   instKP8BtnAct.old.kp8Config[29].activate[5] := TRUE;
   instKP8BtnAct.old.kp8Config[29].activate[6] := TRUE;
   instKP8BtnAct.old.kp8Config[29].activate[7] := TRUE;
   instKP8BtnAct.old.kp8Config[29].colorOn1[0] := 'off';
   instKP8BtnAct.old.kp8Config[29].colorOn1[1] := 'yellow';
   instKP8BtnAct.old.kp8Config[29].colorOn1[2] := 'yellow';
   instKP8BtnAct.old.kp8Config[29].colorOn1[3] := 'yellow';
   instKP8BtnAct.old.kp8Config[29].colorOn1[4] := 'off';
   instKP8BtnAct.old.kp8Config[29].colorOn1[5] := 'yellow';
   instKP8BtnAct.old.kp8Config[29].colorOn1[6] := 'yellow';
   instKP8BtnAct.old.kp8Config[29].colorOn1[7] := 'yellow';
   instKP8BtnAct.old.kp8Config[29].colorOn2[0] := 'off';
   instKP8BtnAct.old.kp8Config[29].colorOn2[4] := 'off';
   instKP8BtnAct.old.kp8Config[29].colorOff[0] := 'off';
   instKP8BtnAct.old.kp8Config[29].colorOff[1] := 'green';
   instKP8BtnAct.old.kp8Config[29].colorOff[2] := 'green';
   instKP8BtnAct.old.kp8Config[29].colorOff[3] := 'green';
   instKP8BtnAct.old.kp8Config[29].colorOff[4] := 'off';
   instKP8BtnAct.old.kp8Config[29].colorOff[5] := 'green';
   instKP8BtnAct.old.kp8Config[29].colorOff[6] := 'green';
   instKP8BtnAct.old.kp8Config[29].colorOff[7] := 'green';
   instKP8BtnAct.old.kp8Config[29].mode[1] := TRUE;
   instKP8BtnAct.old.kp8Config[29].mode[2] := TRUE;
   instKP8BtnAct.old.kp8Config[29].mode[3] := TRUE;
   instKP8BtnAct.old.kp8Config[29].mode[5] := TRUE;
   instKP8BtnAct.old.kp8Config[29].mode[6] := TRUE;
   instKP8BtnAct.old.kp8Config[29].mode[7] := TRUE;
   instKP8BtnAct.old.kp8Config[30].activate[7] := TRUE;
   instKP8BtnAct.old.kp8Config[30].colorOn1[0] := 'off';
   instKP8BtnAct.old.kp8Config[30].colorOn1[1] := 'off';
   instKP8BtnAct.old.kp8Config[30].colorOn1[2] := 'off';
   instKP8BtnAct.old.kp8Config[30].colorOn1[3] := 'off';
   instKP8BtnAct.old.kp8Config[30].colorOn1[4] := 'off';
   instKP8BtnAct.old.kp8Config[30].colorOn1[5] := 'off';
   instKP8BtnAct.old.kp8Config[30].colorOn1[6] := 'off';
   instKP8BtnAct.old.kp8Config[30].colorOn1[7] := 'yellow';
   instKP8BtnAct.old.kp8Config[30].colorOn2[0] := 'off';
   instKP8BtnAct.old.kp8Config[30].colorOn2[1] := 'off';
   instKP8BtnAct.old.kp8Config[30].colorOn2[2] := 'off';
   instKP8BtnAct.old.kp8Config[30].colorOn2[3] := 'off';
   instKP8BtnAct.old.kp8Config[30].colorOn2[4] := 'off';
   instKP8BtnAct.old.kp8Config[30].colorOn2[5] := 'off';
   instKP8BtnAct.old.kp8Config[30].colorOn2[6] := 'off';
   instKP8BtnAct.old.kp8Config[30].colorOff[0] := 'off';
   instKP8BtnAct.old.kp8Config[30].colorOff[1] := 'off';
   instKP8BtnAct.old.kp8Config[30].colorOff[2] := 'off';
   instKP8BtnAct.old.kp8Config[30].colorOff[3] := 'off';
   instKP8BtnAct.old.kp8Config[30].colorOff[4] := 'off';
   instKP8BtnAct.old.kp8Config[30].colorOff[5] := 'off';
   instKP8BtnAct.old.kp8Config[30].colorOff[6] := 'off';
   instKP8BtnAct.old.kp8Config[30].colorOff[7] := 'green';
   instKP8BtnAct.old.kp8Config[30].mode[7] := TRUE;
   instKP8BtnAct.old.kp8Config[31].activate[3] := TRUE;
   instKP8BtnAct.old.kp8Config[31].activate[7] := TRUE;
   instKP8BtnAct.old.kp8Config[31].colorOn1[0] := 'off';
   instKP8BtnAct.old.kp8Config[31].colorOn1[1] := 'off';
   instKP8BtnAct.old.kp8Config[31].colorOn1[2] := 'off';
   instKP8BtnAct.old.kp8Config[31].colorOn1[3] := 'yellow';
   instKP8BtnAct.old.kp8Config[31].colorOn1[4] := 'off';
   instKP8BtnAct.old.kp8Config[31].colorOn1[5] := 'off';
   instKP8BtnAct.old.kp8Config[31].colorOn1[6] := 'off';
   instKP8BtnAct.old.kp8Config[31].colorOn1[7] := 'yellow';
   instKP8BtnAct.old.kp8Config[31].colorOn2[0] := 'off';
   instKP8BtnAct.old.kp8Config[31].colorOn2[1] := 'off';
   instKP8BtnAct.old.kp8Config[31].colorOn2[2] := 'off';
   instKP8BtnAct.old.kp8Config[31].colorOn2[4] := 'off';
   instKP8BtnAct.old.kp8Config[31].colorOn2[5] := 'off';
   instKP8BtnAct.old.kp8Config[31].colorOn2[6] := 'off';
   instKP8BtnAct.old.kp8Config[31].colorOff[0] := 'off';
   instKP8BtnAct.old.kp8Config[31].colorOff[1] := 'off';
   instKP8BtnAct.old.kp8Config[31].colorOff[2] := 'off';
   instKP8BtnAct.old.kp8Config[31].colorOff[3] := 'green';
   instKP8BtnAct.old.kp8Config[31].colorOff[4] := 'off';
   instKP8BtnAct.old.kp8Config[31].colorOff[5] := 'off';
   instKP8BtnAct.old.kp8Config[31].colorOff[6] := 'off';
   instKP8BtnAct.old.kp8Config[31].colorOff[7] := 'green';
   instKP8BtnAct.old.kp8Config[31].mode[3] := TRUE;
   instKP8BtnAct.old.kp8Config[31].mode[7] := TRUE;
   instKP8BtnAct.old.kp8Config[32].activate[7] := TRUE;
   instKP8BtnAct.old.kp8Config[32].colorOn1[0] := 'off';
   instKP8BtnAct.old.kp8Config[32].colorOn1[1] := 'off';
   instKP8BtnAct.old.kp8Config[32].colorOn1[2] := 'off';
   instKP8BtnAct.old.kp8Config[32].colorOn1[3] := 'off';
   instKP8BtnAct.old.kp8Config[32].colorOn1[4] := 'off';
   instKP8BtnAct.old.kp8Config[32].colorOn1[5] := 'off';
   instKP8BtnAct.old.kp8Config[32].colorOn1[6] := 'off';
   instKP8BtnAct.old.kp8Config[32].colorOn1[7] := 'yellow';
   instKP8BtnAct.old.kp8Config[32].colorOn2[0] := 'off';
   instKP8BtnAct.old.kp8Config[32].colorOn2[1] := 'off';
   instKP8BtnAct.old.kp8Config[32].colorOn2[2] := 'off';
   instKP8BtnAct.old.kp8Config[32].colorOn2[3] := 'off';
   instKP8BtnAct.old.kp8Config[32].colorOn2[4] := 'off';
   instKP8BtnAct.old.kp8Config[32].colorOn2[5] := 'off';
   instKP8BtnAct.old.kp8Config[32].colorOn2[6] := 'off';
   instKP8BtnAct.old.kp8Config[32].colorOff[0] := 'off';
   instKP8BtnAct.old.kp8Config[32].colorOff[1] := 'off';
   instKP8BtnAct.old.kp8Config[32].colorOff[2] := 'off';
   instKP8BtnAct.old.kp8Config[32].colorOff[3] := 'off';
   instKP8BtnAct.old.kp8Config[32].colorOff[4] := 'off';
   instKP8BtnAct.old.kp8Config[32].colorOff[5] := 'off';
   instKP8BtnAct.old.kp8Config[32].colorOff[6] := 'off';
   instKP8BtnAct.old.kp8Config[32].colorOff[7] := 'green';
   instKP8BtnAct.old.kp8Config[32].mode[7] := TRUE;
   instKP8BtnAct.old.kp8Config[33].activate[7] := TRUE;
   instKP8BtnAct.old.kp8Config[33].colorOn1[0] := 'off';
   instKP8BtnAct.old.kp8Config[33].colorOn1[1] := 'off';
   instKP8BtnAct.old.kp8Config[33].colorOn1[2] := 'off';
   instKP8BtnAct.old.kp8Config[33].colorOn1[3] := 'off';
   instKP8BtnAct.old.kp8Config[33].colorOn1[4] := 'off';
   instKP8BtnAct.old.kp8Config[33].colorOn1[5] := 'off';
   instKP8BtnAct.old.kp8Config[33].colorOn1[6] := 'off';
   instKP8BtnAct.old.kp8Config[33].colorOn1[7] := 'yellow';
   instKP8BtnAct.old.kp8Config[33].colorOn2[0] := 'off';
   instKP8BtnAct.old.kp8Config[33].colorOn2[1] := 'off';
   instKP8BtnAct.old.kp8Config[33].colorOn2[2] := 'off';
   instKP8BtnAct.old.kp8Config[33].colorOn2[3] := 'off';
   instKP8BtnAct.old.kp8Config[33].colorOn2[4] := 'off';
   instKP8BtnAct.old.kp8Config[33].colorOn2[5] := 'off';
   instKP8BtnAct.old.kp8Config[33].colorOn2[6] := 'off';
   instKP8BtnAct.old.kp8Config[33].colorOff[0] := 'off';
   instKP8BtnAct.old.kp8Config[33].colorOff[1] := 'off';
   instKP8BtnAct.old.kp8Config[33].colorOff[2] := 'off';
   instKP8BtnAct.old.kp8Config[33].colorOff[3] := 'off';
   instKP8BtnAct.old.kp8Config[33].colorOff[4] := 'off';
   instKP8BtnAct.old.kp8Config[33].colorOff[5] := 'off';
   instKP8BtnAct.old.kp8Config[33].colorOff[6] := 'off';
   instKP8BtnAct.old.kp8Config[33].colorOff[7] := 'green';
   instKP8BtnAct.old.kp8Config[33].mode[7] := TRUE;
   instKP8BtnAct.old.kp8Config[34].activate[3] := TRUE;
   instKP8BtnAct.old.kp8Config[34].activate[7] := TRUE;
   instKP8BtnAct.old.kp8Config[34].colorOn1[0] := 'off';
   instKP8BtnAct.old.kp8Config[34].colorOn1[1] := 'off';
   instKP8BtnAct.old.kp8Config[34].colorOn1[2] := 'off';
   instKP8BtnAct.old.kp8Config[34].colorOn1[3] := 'yellow';
   instKP8BtnAct.old.kp8Config[34].colorOn1[4] := 'off';
   instKP8BtnAct.old.kp8Config[34].colorOn1[5] := 'off';
   instKP8BtnAct.old.kp8Config[34].colorOn1[6] := 'off';
   instKP8BtnAct.old.kp8Config[34].colorOn1[7] := 'yellow';
   instKP8BtnAct.old.kp8Config[34].colorOn2[0] := 'off';
   instKP8BtnAct.old.kp8Config[34].colorOn2[1] := 'off';
   instKP8BtnAct.old.kp8Config[34].colorOn2[2] := 'off';
   instKP8BtnAct.old.kp8Config[34].colorOn2[4] := 'off';
   instKP8BtnAct.old.kp8Config[34].colorOn2[5] := 'off';
   instKP8BtnAct.old.kp8Config[34].colorOn2[6] := 'off';
   instKP8BtnAct.old.kp8Config[34].colorOff[0] := 'off';
   instKP8BtnAct.old.kp8Config[34].colorOff[1] := 'off';
   instKP8BtnAct.old.kp8Config[34].colorOff[2] := 'off';
   instKP8BtnAct.old.kp8Config[34].colorOff[3] := 'green';
   instKP8BtnAct.old.kp8Config[34].colorOff[4] := 'off';
   instKP8BtnAct.old.kp8Config[34].colorOff[5] := 'off';
   instKP8BtnAct.old.kp8Config[34].colorOff[6] := 'off';
   instKP8BtnAct.old.kp8Config[34].colorOff[7] := 'green';
   instKP8BtnAct.old.kp8Config[34].mode[3] := TRUE;
   instKP8BtnAct.old.kp8Config[34].mode[7] := TRUE;
   instKP8BtnAct.old.kp8Config[35].activate[3] := TRUE;
   instKP8BtnAct.old.kp8Config[35].activate[7] := TRUE;
   instKP8BtnAct.old.kp8Config[35].colorOn1[0] := 'off';
   instKP8BtnAct.old.kp8Config[35].colorOn1[1] := 'off';
   instKP8BtnAct.old.kp8Config[35].colorOn1[2] := 'off';
   instKP8BtnAct.old.kp8Config[35].colorOn1[3] := 'yellow';
   instKP8BtnAct.old.kp8Config[35].colorOn1[4] := 'off';
   instKP8BtnAct.old.kp8Config[35].colorOn1[5] := 'off';
   instKP8BtnAct.old.kp8Config[35].colorOn1[6] := 'off';
   instKP8BtnAct.old.kp8Config[35].colorOn1[7] := 'yellow';
   instKP8BtnAct.old.kp8Config[35].colorOn2[0] := 'off';
   instKP8BtnAct.old.kp8Config[35].colorOn2[1] := 'off';
   instKP8BtnAct.old.kp8Config[35].colorOn2[2] := 'off';
   instKP8BtnAct.old.kp8Config[35].colorOn2[4] := 'off';
   instKP8BtnAct.old.kp8Config[35].colorOn2[5] := 'off';
   instKP8BtnAct.old.kp8Config[35].colorOn2[6] := 'off';
   instKP8BtnAct.old.kp8Config[35].colorOff[0] := 'off';
   instKP8BtnAct.old.kp8Config[35].colorOff[1] := 'off';
   instKP8BtnAct.old.kp8Config[35].colorOff[2] := 'off';
   instKP8BtnAct.old.kp8Config[35].colorOff[3] := 'green';
   instKP8BtnAct.old.kp8Config[35].colorOff[4] := 'off';
   instKP8BtnAct.old.kp8Config[35].colorOff[5] := 'off';
   instKP8BtnAct.old.kp8Config[35].colorOff[6] := 'off';
   instKP8BtnAct.old.kp8Config[35].colorOff[7] := 'green';
   instKP8BtnAct.old.kp8Config[35].mode[3] := TRUE;
   instKP8BtnAct.old.kp8Config[35].mode[7] := TRUE;
   instKP8BtnAct.old.kp8Config[36].activate[3] := TRUE;
   instKP8BtnAct.old.kp8Config[36].activate[7] := TRUE;
   instKP8BtnAct.old.kp8Config[36].colorOn1[0] := 'off';
   instKP8BtnAct.old.kp8Config[36].colorOn1[1] := 'off';
   instKP8BtnAct.old.kp8Config[36].colorOn1[2] := 'off';
   instKP8BtnAct.old.kp8Config[36].colorOn1[3] := 'yellow';
   instKP8BtnAct.old.kp8Config[36].colorOn1[4] := 'off';
   instKP8BtnAct.old.kp8Config[36].colorOn1[5] := 'off';
   instKP8BtnAct.old.kp8Config[36].colorOn1[6] := 'off';
   instKP8BtnAct.old.kp8Config[36].colorOn1[7] := 'yellow';
   instKP8BtnAct.old.kp8Config[36].colorOn2[0] := 'off';
   instKP8BtnAct.old.kp8Config[36].colorOn2[1] := 'off';
   instKP8BtnAct.old.kp8Config[36].colorOn2[2] := 'off';
   instKP8BtnAct.old.kp8Config[36].colorOn2[4] := 'off';
   instKP8BtnAct.old.kp8Config[36].colorOn2[5] := 'off';
   instKP8BtnAct.old.kp8Config[36].colorOn2[6] := 'off';
   instKP8BtnAct.old.kp8Config[36].colorOff[0] := 'off';
   instKP8BtnAct.old.kp8Config[36].colorOff[1] := 'off';
   instKP8BtnAct.old.kp8Config[36].colorOff[2] := 'off';
   instKP8BtnAct.old.kp8Config[36].colorOff[3] := 'green';
   instKP8BtnAct.old.kp8Config[36].colorOff[4] := 'off';
   instKP8BtnAct.old.kp8Config[36].colorOff[5] := 'off';
   instKP8BtnAct.old.kp8Config[36].colorOff[6] := 'off';
   instKP8BtnAct.old.kp8Config[36].colorOff[7] := 'green';
   instKP8BtnAct.old.kp8Config[36].mode[3] := TRUE;
   instKP8BtnAct.old.kp8Config[36].mode[7] := TRUE;
   instKP8BtnAct.old.kp8Config[37].activate[3] := TRUE;
   instKP8BtnAct.old.kp8Config[37].activate[7] := TRUE;
   instKP8BtnAct.old.kp8Config[37].colorOn1[0] := 'off';
   instKP8BtnAct.old.kp8Config[37].colorOn1[1] := 'off';
   instKP8BtnAct.old.kp8Config[37].colorOn1[2] := 'off';
   instKP8BtnAct.old.kp8Config[37].colorOn1[3] := 'yellow';
   instKP8BtnAct.old.kp8Config[37].colorOn1[4] := 'off';
   instKP8BtnAct.old.kp8Config[37].colorOn1[5] := 'off';
   instKP8BtnAct.old.kp8Config[37].colorOn1[6] := 'off';
   instKP8BtnAct.old.kp8Config[37].colorOn1[7] := 'yellow';
   instKP8BtnAct.old.kp8Config[37].colorOn2[0] := 'off';
   instKP8BtnAct.old.kp8Config[37].colorOn2[1] := 'off';
   instKP8BtnAct.old.kp8Config[37].colorOn2[2] := 'off';
   instKP8BtnAct.old.kp8Config[37].colorOn2[4] := 'off';
   instKP8BtnAct.old.kp8Config[37].colorOn2[5] := 'off';
   instKP8BtnAct.old.kp8Config[37].colorOn2[6] := 'off';
   instKP8BtnAct.old.kp8Config[37].colorOff[0] := 'off';
   instKP8BtnAct.old.kp8Config[37].colorOff[1] := 'off';
   instKP8BtnAct.old.kp8Config[37].colorOff[2] := 'off';
   instKP8BtnAct.old.kp8Config[37].colorOff[3] := 'green';
   instKP8BtnAct.old.kp8Config[37].colorOff[4] := 'off';
   instKP8BtnAct.old.kp8Config[37].colorOff[5] := 'off';
   instKP8BtnAct.old.kp8Config[37].colorOff[6] := 'off';
   instKP8BtnAct.old.kp8Config[37].colorOff[7] := 'green';
   instKP8BtnAct.old.kp8Config[37].mode[3] := TRUE;
   instKP8BtnAct.old.kp8Config[37].mode[7] := TRUE;
   instKP8BtnAct.old.kp8Config[38].activate[7] := TRUE;
   instKP8BtnAct.old.kp8Config[38].colorOn1[0] := 'off';
   instKP8BtnAct.old.kp8Config[38].colorOn1[1] := 'off';
   instKP8BtnAct.old.kp8Config[38].colorOn1[2] := 'off';
   instKP8BtnAct.old.kp8Config[38].colorOn1[3] := 'off';
   instKP8BtnAct.old.kp8Config[38].colorOn1[4] := 'off';
   instKP8BtnAct.old.kp8Config[38].colorOn1[5] := 'off';
   instKP8BtnAct.old.kp8Config[38].colorOn1[6] := 'off';
   instKP8BtnAct.old.kp8Config[38].colorOn1[7] := 'yellow';
   instKP8BtnAct.old.kp8Config[38].colorOn2[0] := 'off';
   instKP8BtnAct.old.kp8Config[38].colorOn2[1] := 'off';
   instKP8BtnAct.old.kp8Config[38].colorOn2[2] := 'off';
   instKP8BtnAct.old.kp8Config[38].colorOn2[3] := 'off';
   instKP8BtnAct.old.kp8Config[38].colorOn2[4] := 'off';
   instKP8BtnAct.old.kp8Config[38].colorOn2[5] := 'off';
   instKP8BtnAct.old.kp8Config[38].colorOn2[6] := 'off';
   instKP8BtnAct.old.kp8Config[38].colorOff[0] := 'off';
   instKP8BtnAct.old.kp8Config[38].colorOff[1] := 'off';
   instKP8BtnAct.old.kp8Config[38].colorOff[2] := 'off';
   instKP8BtnAct.old.kp8Config[38].colorOff[3] := 'off';
   instKP8BtnAct.old.kp8Config[38].colorOff[4] := 'off';
   instKP8BtnAct.old.kp8Config[38].colorOff[5] := 'off';
   instKP8BtnAct.old.kp8Config[38].colorOff[6] := 'off';
   instKP8BtnAct.old.kp8Config[38].colorOff[7] := 'green';
   instKP8BtnAct.old.kp8Config[38].mode[7] := TRUE;
   instKP8Drvs[0].btn0ColorOn1 := 'off';
   instKP8Drvs[0].btn0ColorOn2 := 'off';
   instKP8Drvs[0].btn0ColorOff := 'off';
   instKP8Drvs[0].btn1ColorOn1 := 'off';
   instKP8Drvs[0].btn1ColorOn2 := 'off';
   instKP8Drvs[0].btn1ColorOff := 'off';
   instKP8Drvs[0].btn2ColorOn1 := 'off';
   instKP8Drvs[0].btn2ColorOn2 := 'off';
   instKP8Drvs[0].btn2ColorOff := 'off';
   instKP8Drvs[0].btn3Activate := TRUE;
   instKP8Drvs[0].btn3Mode := TRUE;
   instKP8Drvs[0].btn3ColorOn1 := 'yellow';
   instKP8Drvs[0].btn3ColorOff := 'green';
   instKP8Drvs[0].btn4ColorOn1 := 'off';
   instKP8Drvs[0].btn4ColorOn2 := 'off';
   instKP8Drvs[0].btn4ColorOff := 'off';
   instKP8Drvs[0].btn5ColorOn1 := 'off';
   instKP8Drvs[0].btn5ColorOn2 := 'off';
   instKP8Drvs[0].btn5ColorOff := 'off';
   instKP8Drvs[0].btn6ColorOn1 := 'off';
   instKP8Drvs[0].btn6ColorOn2 := 'off';
   instKP8Drvs[0].btn6ColorOff := 'off';
   instKP8Drvs[0].btn7Activate := TRUE;
   instKP8Drvs[0].btn7Mode := TRUE;
   instKP8Drvs[0].btn7ColorOn1 := 'yellow';
   instKP8Drvs[0].btn7ColorOff := 'green';
   instKP8Drvs[0].btnColorsOut := 16#0088_0000;
   instKP8Drvs[0].i1 := 8;
   instKP8Drvs[0].i2 := 8;
   instKP8Drvs[0].btnActivateInt[3] := TRUE;
   instKP8Drvs[0].btnActivateInt[7] := TRUE;
   instKP8Drvs[0].btnClrMskOffInt[0] := 16#0000_0000;
   instKP8Drvs[0].btnClrMskOffInt[1] := 16#0000_0000;
   instKP8Drvs[0].btnClrMskOffInt[2] := 16#0000_0000;
   instKP8Drvs[0].btnClrMskOffInt[3] := 16#0008_0000;
   instKP8Drvs[0].btnClrMskOffInt[4] := 16#0000_0000;
   instKP8Drvs[0].btnClrMskOffInt[5] := 16#0000_0000;
   instKP8Drvs[0].btnClrMskOffInt[6] := 16#0000_0000;
   instKP8Drvs[0].btnClrMskOffInt[7] := 16#0080_0000;
   instKP8Drvs[0].btnClrMskOn1Int[0] := 16#0000_0000;
   instKP8Drvs[0].btnClrMskOn1Int[1] := 16#0000_0000;
   instKP8Drvs[0].btnClrMskOn1Int[2] := 16#0000_0000;
   instKP8Drvs[0].btnClrMskOn1Int[3] := 16#0808_0000;
   instKP8Drvs[0].btnClrMskOn1Int[4] := 16#0000_0000;
   instKP8Drvs[0].btnClrMskOn1Int[5] := 16#0000_0000;
   instKP8Drvs[0].btnClrMskOn1Int[6] := 16#0000_0000;
   instKP8Drvs[0].btnClrMskOn1Int[7] := 16#8080_0000;
   instKP8Drvs[0].btnClrMskOn2Int[0] := 16#0000_0000;
   instKP8Drvs[0].btnClrMskOn2Int[1] := 16#0000_0000;
   instKP8Drvs[0].btnClrMskOn2Int[2] := 16#0000_0000;
   instKP8Drvs[0].btnClrMskOn2Int[3] := 16#0000_0000;
   instKP8Drvs[0].btnClrMskOn2Int[4] := 16#0000_0000;
   instKP8Drvs[0].btnClrMskOn2Int[5] := 16#0000_0000;
   instKP8Drvs[0].btnClrMskOn2Int[6] := 16#0000_0000;
   instKP8Drvs[0].btnClrMskOn2Int[7] := 16#0000_0000;
   instKP8Drvs[0].btnClrOffInt[0] := 'off';
   instKP8Drvs[0].btnClrOffInt[1] := 'off';
   instKP8Drvs[0].btnClrOffInt[2] := 'off';
   instKP8Drvs[0].btnClrOffInt[3] := 'green';
   instKP8Drvs[0].btnClrOffInt[4] := 'off';
   instKP8Drvs[0].btnClrOffInt[5] := 'off';
   instKP8Drvs[0].btnClrOffInt[6] := 'off';
   instKP8Drvs[0].btnClrOffInt[7] := 'green';
   instKP8Drvs[0].btnClrOn1Int[0] := 'off';
   instKP8Drvs[0].btnClrOn1Int[1] := 'off';
   instKP8Drvs[0].btnClrOn1Int[2] := 'off';
   instKP8Drvs[0].btnClrOn1Int[3] := 'yellow';
   instKP8Drvs[0].btnClrOn1Int[4] := 'off';
   instKP8Drvs[0].btnClrOn1Int[5] := 'off';
   instKP8Drvs[0].btnClrOn1Int[6] := 'off';
   instKP8Drvs[0].btnClrOn1Int[7] := 'yellow';
   instKP8Drvs[0].btnClrOn2Int[0] := 'off';
   instKP8Drvs[0].btnClrOn2Int[1] := 'off';
   instKP8Drvs[0].btnClrOn2Int[2] := 'off';
   instKP8Drvs[0].btnClrOn2Int[4] := 'off';
   instKP8Drvs[0].btnClrOn2Int[5] := 'off';
   instKP8Drvs[0].btnClrOn2Int[6] := 'off';
   instKP8Drvs[0].btnColors := 16#0088_0000;
   instKP8Drvs[0].btnModeInt[3] := TRUE;
   instKP8Drvs[0].btnModeInt[7] := TRUE;
   instKP8Drvs[1].btn0ColorOn1 := 'off';
   instKP8Drvs[1].btn0ColorOn2 := 'off';
   instKP8Drvs[1].btn0ColorOff := 'off';
   instKP8Drvs[1].btn1ColorOn1 := 'off';
   instKP8Drvs[1].btn1ColorOn2 := 'off';
   instKP8Drvs[1].btn1ColorOff := 'off';
   instKP8Drvs[1].btn2Activate := TRUE;
   instKP8Drvs[1].btn2Mode := TRUE;
   instKP8Drvs[1].btn2ColorOn1 := 'yellow';
   instKP8Drvs[1].btn2ColorOff := 'green';
   instKP8Drvs[1].btn3Activate := TRUE;
   instKP8Drvs[1].btn3Mode := TRUE;
   instKP8Drvs[1].btn3ColorOn1 := 'yellow';
   instKP8Drvs[1].btn3ColorOff := 'green';
   instKP8Drvs[1].btn4ColorOn1 := 'off';
   instKP8Drvs[1].btn4ColorOn2 := 'off';
   instKP8Drvs[1].btn4ColorOff := 'off';
   instKP8Drvs[1].btn5ColorOn1 := 'off';
   instKP8Drvs[1].btn5ColorOn2 := 'off';
   instKP8Drvs[1].btn5ColorOff := 'off';
   instKP8Drvs[1].btn6Activate := TRUE;
   instKP8Drvs[1].btn6Mode := TRUE;
   instKP8Drvs[1].btn6ColorOn1 := 'yellow';
   instKP8Drvs[1].btn6ColorOff := 'green';
   instKP8Drvs[1].btn7Activate := TRUE;
   instKP8Drvs[1].btn7Mode := TRUE;
   instKP8Drvs[1].btn7ColorOn1 := 'yellow';
   instKP8Drvs[1].btn7ColorOff := 'green';
   instKP8Drvs[1].btnColorsOut := 16#00CC_0000;
   instKP8Drvs[1].i1 := 8;
   instKP8Drvs[1].i2 := 8;
   instKP8Drvs[1].btnActivateInt[2] := TRUE;
   instKP8Drvs[1].btnActivateInt[3] := TRUE;
   instKP8Drvs[1].btnActivateInt[6] := TRUE;
   instKP8Drvs[1].btnActivateInt[7] := TRUE;
   instKP8Drvs[1].btnClrMskOffInt[0] := 16#0000_0000;
   instKP8Drvs[1].btnClrMskOffInt[1] := 16#0000_0000;
   instKP8Drvs[1].btnClrMskOffInt[2] := 16#0004_0000;
   instKP8Drvs[1].btnClrMskOffInt[3] := 16#0008_0000;
   instKP8Drvs[1].btnClrMskOffInt[4] := 16#0000_0000;
   instKP8Drvs[1].btnClrMskOffInt[5] := 16#0000_0000;
   instKP8Drvs[1].btnClrMskOffInt[6] := 16#0040_0000;
   instKP8Drvs[1].btnClrMskOffInt[7] := 16#0080_0000;
   instKP8Drvs[1].btnClrMskOn1Int[0] := 16#0000_0000;
   instKP8Drvs[1].btnClrMskOn1Int[1] := 16#0000_0000;
   instKP8Drvs[1].btnClrMskOn1Int[2] := 16#0404_0000;
   instKP8Drvs[1].btnClrMskOn1Int[3] := 16#0808_0000;
   instKP8Drvs[1].btnClrMskOn1Int[4] := 16#0000_0000;
   instKP8Drvs[1].btnClrMskOn1Int[5] := 16#0000_0000;
   instKP8Drvs[1].btnClrMskOn1Int[6] := 16#4040_0000;
   instKP8Drvs[1].btnClrMskOn1Int[7] := 16#8080_0000;
   instKP8Drvs[1].btnClrMskOn2Int[0] := 16#0000_0000;
   instKP8Drvs[1].btnClrMskOn2Int[1] := 16#0000_0000;
   instKP8Drvs[1].btnClrMskOn2Int[2] := 16#0000_0000;
   instKP8Drvs[1].btnClrMskOn2Int[3] := 16#0000_0000;
   instKP8Drvs[1].btnClrMskOn2Int[4] := 16#0000_0000;
   instKP8Drvs[1].btnClrMskOn2Int[5] := 16#0000_0000;
   instKP8Drvs[1].btnClrMskOn2Int[6] := 16#0000_0000;
   instKP8Drvs[1].btnClrMskOn2Int[7] := 16#0000_0000;
   instKP8Drvs[1].btnClrOffInt[0] := 'off';
   instKP8Drvs[1].btnClrOffInt[1] := 'off';
   instKP8Drvs[1].btnClrOffInt[2] := 'green';
   instKP8Drvs[1].btnClrOffInt[3] := 'green';
   instKP8Drvs[1].btnClrOffInt[4] := 'off';
   instKP8Drvs[1].btnClrOffInt[5] := 'off';
   instKP8Drvs[1].btnClrOffInt[6] := 'green';
   instKP8Drvs[1].btnClrOffInt[7] := 'green';
   instKP8Drvs[1].btnClrOn1Int[0] := 'off';
   instKP8Drvs[1].btnClrOn1Int[1] := 'off';
   instKP8Drvs[1].btnClrOn1Int[2] := 'yellow';
   instKP8Drvs[1].btnClrOn1Int[3] := 'yellow';
   instKP8Drvs[1].btnClrOn1Int[4] := 'off';
   instKP8Drvs[1].btnClrOn1Int[5] := 'off';
   instKP8Drvs[1].btnClrOn1Int[6] := 'yellow';
   instKP8Drvs[1].btnClrOn1Int[7] := 'yellow';
   instKP8Drvs[1].btnClrOn2Int[0] := 'off';
   instKP8Drvs[1].btnClrOn2Int[1] := 'off';
   instKP8Drvs[1].btnClrOn2Int[4] := 'off';
   instKP8Drvs[1].btnClrOn2Int[5] := 'off';
   instKP8Drvs[1].btnColors := 16#00CC_0000;
   instKP8Drvs[1].btnModeInt[2] := TRUE;
   instKP8Drvs[1].btnModeInt[3] := TRUE;
   instKP8Drvs[1].btnModeInt[6] := TRUE;
   instKP8Drvs[1].btnModeInt[7] := TRUE;
   instKP8Drvs[2].btn0ColorOn1 := 'off';
   instKP8Drvs[2].btn0ColorOn2 := 'off';
   instKP8Drvs[2].btn0ColorOff := 'off';
   instKP8Drvs[2].btn1Activate := TRUE;
   instKP8Drvs[2].btn1Mode := TRUE;
   instKP8Drvs[2].btn1ColorOn1 := 'yellow';
   instKP8Drvs[2].btn1ColorOff := 'green';
   instKP8Drvs[2].btn2Activate := TRUE;
   instKP8Drvs[2].btn2Mode := TRUE;
   instKP8Drvs[2].btn2ColorOn1 := 'yellow';
   instKP8Drvs[2].btn2ColorOff := 'green';
   instKP8Drvs[2].btn3Activate := TRUE;
   instKP8Drvs[2].btn3Mode := TRUE;
   instKP8Drvs[2].btn3ColorOn1 := 'yellow';
   instKP8Drvs[2].btn3ColorOff := 'green';
   instKP8Drvs[2].btn4ColorOn1 := 'off';
   instKP8Drvs[2].btn4ColorOn2 := 'off';
   instKP8Drvs[2].btn4ColorOff := 'off';
   instKP8Drvs[2].btn5Activate := TRUE;
   instKP8Drvs[2].btn5Mode := TRUE;
   instKP8Drvs[2].btn5ColorOn1 := 'yellow';
   instKP8Drvs[2].btn5ColorOff := 'green';
   instKP8Drvs[2].btn6Activate := TRUE;
   instKP8Drvs[2].btn6Mode := TRUE;
   instKP8Drvs[2].btn6ColorOn1 := 'yellow';
   instKP8Drvs[2].btn6ColorOff := 'green';
   instKP8Drvs[2].btn7Activate := TRUE;
   instKP8Drvs[2].btn7Mode := TRUE;
   instKP8Drvs[2].btn7ColorOn1 := 'yellow';
   instKP8Drvs[2].btn7ColorOff := 'green';
   instKP8Drvs[2].btnColorsOut := 16#00EE_0000;
   instKP8Drvs[2].i1 := 8;
   instKP8Drvs[2].i2 := 8;
   instKP8Drvs[2].btnActivateInt[1] := TRUE;
   instKP8Drvs[2].btnActivateInt[2] := TRUE;
   instKP8Drvs[2].btnActivateInt[3] := TRUE;
   instKP8Drvs[2].btnActivateInt[5] := TRUE;
   instKP8Drvs[2].btnActivateInt[6] := TRUE;
   instKP8Drvs[2].btnActivateInt[7] := TRUE;
   instKP8Drvs[2].btnClrMskOffInt[0] := 16#0000_0000;
   instKP8Drvs[2].btnClrMskOffInt[1] := 16#0002_0000;
   instKP8Drvs[2].btnClrMskOffInt[2] := 16#0004_0000;
   instKP8Drvs[2].btnClrMskOffInt[3] := 16#0008_0000;
   instKP8Drvs[2].btnClrMskOffInt[4] := 16#0000_0000;
   instKP8Drvs[2].btnClrMskOffInt[5] := 16#0020_0000;
   instKP8Drvs[2].btnClrMskOffInt[6] := 16#0040_0000;
   instKP8Drvs[2].btnClrMskOffInt[7] := 16#0080_0000;
   instKP8Drvs[2].btnClrMskOn1Int[0] := 16#0000_0000;
   instKP8Drvs[2].btnClrMskOn1Int[1] := 16#0202_0000;
   instKP8Drvs[2].btnClrMskOn1Int[2] := 16#0404_0000;
   instKP8Drvs[2].btnClrMskOn1Int[3] := 16#0808_0000;
   instKP8Drvs[2].btnClrMskOn1Int[4] := 16#0000_0000;
   instKP8Drvs[2].btnClrMskOn1Int[5] := 16#2020_0000;
   instKP8Drvs[2].btnClrMskOn1Int[6] := 16#4040_0000;
   instKP8Drvs[2].btnClrMskOn1Int[7] := 16#8080_0000;
   instKP8Drvs[2].btnClrMskOn2Int[0] := 16#0000_0000;
   instKP8Drvs[2].btnClrMskOn2Int[1] := 16#0000_0000;
   instKP8Drvs[2].btnClrMskOn2Int[2] := 16#0000_0000;
   instKP8Drvs[2].btnClrMskOn2Int[3] := 16#0000_0000;
   instKP8Drvs[2].btnClrMskOn2Int[4] := 16#0000_0000;
   instKP8Drvs[2].btnClrMskOn2Int[5] := 16#0000_0000;
   instKP8Drvs[2].btnClrMskOn2Int[6] := 16#0000_0000;
   instKP8Drvs[2].btnClrMskOn2Int[7] := 16#0000_0000;
   instKP8Drvs[2].btnClrOffInt[0] := 'off';
   instKP8Drvs[2].btnClrOffInt[1] := 'green';
   instKP8Drvs[2].btnClrOffInt[2] := 'green';
   instKP8Drvs[2].btnClrOffInt[3] := 'green';
   instKP8Drvs[2].btnClrOffInt[4] := 'off';
   instKP8Drvs[2].btnClrOffInt[5] := 'green';
   instKP8Drvs[2].btnClrOffInt[6] := 'green';
   instKP8Drvs[2].btnClrOffInt[7] := 'green';
   instKP8Drvs[2].btnClrOn1Int[0] := 'off';
   instKP8Drvs[2].btnClrOn1Int[1] := 'yellow';
   instKP8Drvs[2].btnClrOn1Int[2] := 'yellow';
   instKP8Drvs[2].btnClrOn1Int[3] := 'yellow';
   instKP8Drvs[2].btnClrOn1Int[4] := 'off';
   instKP8Drvs[2].btnClrOn1Int[5] := 'yellow';
   instKP8Drvs[2].btnClrOn1Int[6] := 'yellow';
   instKP8Drvs[2].btnClrOn1Int[7] := 'yellow';
   instKP8Drvs[2].btnClrOn2Int[0] := 'off';
   instKP8Drvs[2].btnClrOn2Int[4] := 'off';
   instKP8Drvs[2].btnColors := 16#00EE_0000;
   instKP8Drvs[2].btnModeInt[1] := TRUE;
   instKP8Drvs[2].btnModeInt[2] := TRUE;
   instKP8Drvs[2].btnModeInt[3] := TRUE;
   instKP8Drvs[2].btnModeInt[5] := TRUE;
   instKP8Drvs[2].btnModeInt[6] := TRUE;
   instKP8Drvs[2].btnModeInt[7] := TRUE;
   instKP8Drvs[3].btn0ColorOn1 := 'off';
   instKP8Drvs[3].btn0ColorOn2 := 'off';
   instKP8Drvs[3].btn0ColorOff := 'off';
   instKP8Drvs[3].btn1Activate := TRUE;
   instKP8Drvs[3].btn1Mode := TRUE;
   instKP8Drvs[3].btn1ColorOn1 := 'yellow';
   instKP8Drvs[3].btn1ColorOff := 'green';
   instKP8Drvs[3].btn2Activate := TRUE;
   instKP8Drvs[3].btn2Mode := TRUE;
   instKP8Drvs[3].btn2ColorOn1 := 'yellow';
   instKP8Drvs[3].btn2ColorOff := 'green';
   instKP8Drvs[3].btn3Activate := TRUE;
   instKP8Drvs[3].btn3Mode := TRUE;
   instKP8Drvs[3].btn3ColorOn1 := 'yellow';
   instKP8Drvs[3].btn3ColorOff := 'green';
   instKP8Drvs[3].btn4ColorOn1 := 'off';
   instKP8Drvs[3].btn4ColorOn2 := 'off';
   instKP8Drvs[3].btn4ColorOff := 'off';
   instKP8Drvs[3].btn5Activate := TRUE;
   instKP8Drvs[3].btn5Mode := TRUE;
   instKP8Drvs[3].btn5ColorOn1 := 'yellow';
   instKP8Drvs[3].btn5ColorOff := 'green';
   instKP8Drvs[3].btn6Activate := TRUE;
   instKP8Drvs[3].btn6Mode := TRUE;
   instKP8Drvs[3].btn6ColorOn1 := 'yellow';
   instKP8Drvs[3].btn6ColorOff := 'green';
   instKP8Drvs[3].btn7Activate := TRUE;
   instKP8Drvs[3].btn7Mode := TRUE;
   instKP8Drvs[3].btn7ColorOn1 := 'yellow';
   instKP8Drvs[3].btn7ColorOff := 'green';
   instKP8Drvs[3].btnColorsOut := 16#00EE_0000;
   instKP8Drvs[3].i1 := 8;
   instKP8Drvs[3].i2 := 8;
   instKP8Drvs[3].btnActivateInt[1] := TRUE;
   instKP8Drvs[3].btnActivateInt[2] := TRUE;
   instKP8Drvs[3].btnActivateInt[3] := TRUE;
   instKP8Drvs[3].btnActivateInt[5] := TRUE;
   instKP8Drvs[3].btnActivateInt[6] := TRUE;
   instKP8Drvs[3].btnActivateInt[7] := TRUE;
   instKP8Drvs[3].btnClrMskOffInt[0] := 16#0000_0000;
   instKP8Drvs[3].btnClrMskOffInt[1] := 16#0002_0000;
   instKP8Drvs[3].btnClrMskOffInt[2] := 16#0004_0000;
   instKP8Drvs[3].btnClrMskOffInt[3] := 16#0008_0000;
   instKP8Drvs[3].btnClrMskOffInt[4] := 16#0000_0000;
   instKP8Drvs[3].btnClrMskOffInt[5] := 16#0020_0000;
   instKP8Drvs[3].btnClrMskOffInt[6] := 16#0040_0000;
   instKP8Drvs[3].btnClrMskOffInt[7] := 16#0080_0000;
   instKP8Drvs[3].btnClrMskOn1Int[0] := 16#0000_0000;
   instKP8Drvs[3].btnClrMskOn1Int[1] := 16#0202_0000;
   instKP8Drvs[3].btnClrMskOn1Int[2] := 16#0404_0000;
   instKP8Drvs[3].btnClrMskOn1Int[3] := 16#0808_0000;
   instKP8Drvs[3].btnClrMskOn1Int[4] := 16#0000_0000;
   instKP8Drvs[3].btnClrMskOn1Int[5] := 16#2020_0000;
   instKP8Drvs[3].btnClrMskOn1Int[6] := 16#4040_0000;
   instKP8Drvs[3].btnClrMskOn1Int[7] := 16#8080_0000;
   instKP8Drvs[3].btnClrMskOn2Int[0] := 16#0000_0000;
   instKP8Drvs[3].btnClrMskOn2Int[1] := 16#0000_0000;
   instKP8Drvs[3].btnClrMskOn2Int[2] := 16#0000_0000;
   instKP8Drvs[3].btnClrMskOn2Int[3] := 16#0000_0000;
   instKP8Drvs[3].btnClrMskOn2Int[4] := 16#0000_0000;
   instKP8Drvs[3].btnClrMskOn2Int[5] := 16#0000_0000;
   instKP8Drvs[3].btnClrMskOn2Int[6] := 16#0000_0000;
   instKP8Drvs[3].btnClrMskOn2Int[7] := 16#0000_0000;
   instKP8Drvs[3].btnClrOffInt[0] := 'off';
   instKP8Drvs[3].btnClrOffInt[1] := 'green';
   instKP8Drvs[3].btnClrOffInt[2] := 'green';
   instKP8Drvs[3].btnClrOffInt[3] := 'green';
   instKP8Drvs[3].btnClrOffInt[4] := 'off';
   instKP8Drvs[3].btnClrOffInt[5] := 'green';
   instKP8Drvs[3].btnClrOffInt[6] := 'green';
   instKP8Drvs[3].btnClrOffInt[7] := 'green';
   instKP8Drvs[3].btnClrOn1Int[0] := 'off';
   instKP8Drvs[3].btnClrOn1Int[1] := 'yellow';
   instKP8Drvs[3].btnClrOn1Int[2] := 'yellow';
   instKP8Drvs[3].btnClrOn1Int[3] := 'yellow';
   instKP8Drvs[3].btnClrOn1Int[4] := 'off';
   instKP8Drvs[3].btnClrOn1Int[5] := 'yellow';
   instKP8Drvs[3].btnClrOn1Int[6] := 'yellow';
   instKP8Drvs[3].btnClrOn1Int[7] := 'yellow';
   instKP8Drvs[3].btnClrOn2Int[0] := 'off';
   instKP8Drvs[3].btnClrOn2Int[4] := 'off';
   instKP8Drvs[3].btnColors := 16#00EE_0000;
   instKP8Drvs[3].btnModeInt[1] := TRUE;
   instKP8Drvs[3].btnModeInt[2] := TRUE;
   instKP8Drvs[3].btnModeInt[3] := TRUE;
   instKP8Drvs[3].btnModeInt[5] := TRUE;
   instKP8Drvs[3].btnModeInt[6] := TRUE;
   instKP8Drvs[3].btnModeInt[7] := TRUE;
   instKP8Drvs[4].btn0ColorOn1 := 'off';
   instKP8Drvs[4].btn0ColorOn2 := 'off';
   instKP8Drvs[4].btn0ColorOff := 'off';
   instKP8Drvs[4].btn1ColorOn1 := 'off';
   instKP8Drvs[4].btn1ColorOn2 := 'off';
   instKP8Drvs[4].btn1ColorOff := 'off';
   instKP8Drvs[4].btn2ColorOn1 := 'off';
   instKP8Drvs[4].btn2ColorOn2 := 'off';
   instKP8Drvs[4].btn2ColorOff := 'off';
   instKP8Drvs[4].btn3ColorOn1 := 'off';
   instKP8Drvs[4].btn3ColorOn2 := 'off';
   instKP8Drvs[4].btn3ColorOff := 'off';
   instKP8Drvs[4].btn4ColorOn1 := 'off';
   instKP8Drvs[4].btn4ColorOn2 := 'off';
   instKP8Drvs[4].btn4ColorOff := 'off';
   instKP8Drvs[4].btn5ColorOn1 := 'off';
   instKP8Drvs[4].btn5ColorOn2 := 'off';
   instKP8Drvs[4].btn5ColorOff := 'off';
   instKP8Drvs[4].btn6ColorOn1 := 'off';
   instKP8Drvs[4].btn6ColorOn2 := 'off';
   instKP8Drvs[4].btn6ColorOff := 'off';
   instKP8Drvs[4].btn7Activate := TRUE;
   instKP8Drvs[4].btn7Mode := TRUE;
   instKP8Drvs[4].btn7ColorOn1 := 'yellow';
   instKP8Drvs[4].btn7ColorOff := 'green';
   instKP8Drvs[4].btnColorsOut := 16#0080_0000;
   instKP8Drvs[4].i1 := 8;
   instKP8Drvs[4].i2 := 8;
   instKP8Drvs[4].btnActivateInt[7] := TRUE;
   instKP8Drvs[4].btnClrMskOffInt[0] := 16#0000_0000;
   instKP8Drvs[4].btnClrMskOffInt[1] := 16#0000_0000;
   instKP8Drvs[4].btnClrMskOffInt[2] := 16#0000_0000;
   instKP8Drvs[4].btnClrMskOffInt[3] := 16#0000_0000;
   instKP8Drvs[4].btnClrMskOffInt[4] := 16#0000_0000;
   instKP8Drvs[4].btnClrMskOffInt[5] := 16#0000_0000;
   instKP8Drvs[4].btnClrMskOffInt[6] := 16#0000_0000;
   instKP8Drvs[4].btnClrMskOffInt[7] := 16#0080_0000;
   instKP8Drvs[4].btnClrMskOn1Int[0] := 16#0000_0000;
   instKP8Drvs[4].btnClrMskOn1Int[1] := 16#0000_0000;
   instKP8Drvs[4].btnClrMskOn1Int[2] := 16#0000_0000;
   instKP8Drvs[4].btnClrMskOn1Int[3] := 16#0000_0000;
   instKP8Drvs[4].btnClrMskOn1Int[4] := 16#0000_0000;
   instKP8Drvs[4].btnClrMskOn1Int[5] := 16#0000_0000;
   instKP8Drvs[4].btnClrMskOn1Int[6] := 16#0000_0000;
   instKP8Drvs[4].btnClrMskOn1Int[7] := 16#8080_0000;
   instKP8Drvs[4].btnClrMskOn2Int[0] := 16#0000_0000;
   instKP8Drvs[4].btnClrMskOn2Int[1] := 16#0000_0000;
   instKP8Drvs[4].btnClrMskOn2Int[2] := 16#0000_0000;
   instKP8Drvs[4].btnClrMskOn2Int[3] := 16#0000_0000;
   instKP8Drvs[4].btnClrMskOn2Int[4] := 16#0000_0000;
   instKP8Drvs[4].btnClrMskOn2Int[5] := 16#0000_0000;
   instKP8Drvs[4].btnClrMskOn2Int[6] := 16#0000_0000;
   instKP8Drvs[4].btnClrMskOn2Int[7] := 16#0000_0000;
   instKP8Drvs[4].btnClrOffInt[0] := 'off';
   instKP8Drvs[4].btnClrOffInt[1] := 'off';
   instKP8Drvs[4].btnClrOffInt[2] := 'off';
   instKP8Drvs[4].btnClrOffInt[3] := 'off';
   instKP8Drvs[4].btnClrOffInt[4] := 'off';
   instKP8Drvs[4].btnClrOffInt[5] := 'off';
   instKP8Drvs[4].btnClrOffInt[6] := 'off';
   instKP8Drvs[4].btnClrOffInt[7] := 'green';
   instKP8Drvs[4].btnClrOn1Int[0] := 'off';
   instKP8Drvs[4].btnClrOn1Int[1] := 'off';
   instKP8Drvs[4].btnClrOn1Int[2] := 'off';
   instKP8Drvs[4].btnClrOn1Int[3] := 'off';
   instKP8Drvs[4].btnClrOn1Int[4] := 'off';
   instKP8Drvs[4].btnClrOn1Int[5] := 'off';
   instKP8Drvs[4].btnClrOn1Int[6] := 'off';
   instKP8Drvs[4].btnClrOn1Int[7] := 'yellow';
   instKP8Drvs[4].btnClrOn2Int[0] := 'off';
   instKP8Drvs[4].btnClrOn2Int[1] := 'off';
   instKP8Drvs[4].btnClrOn2Int[2] := 'off';
   instKP8Drvs[4].btnClrOn2Int[3] := 'off';
   instKP8Drvs[4].btnClrOn2Int[4] := 'off';
   instKP8Drvs[4].btnClrOn2Int[5] := 'off';
   instKP8Drvs[4].btnClrOn2Int[6] := 'off';
   instKP8Drvs[4].btnColors := 16#0080_0000;
   instKP8Drvs[4].btnModeInt[7] := TRUE;
   instKP8Drvs[5].btn0ColorOn1 := 'off';
   instKP8Drvs[5].btn0ColorOn2 := 'off';
   instKP8Drvs[5].btn0ColorOff := 'off';
   instKP8Drvs[5].btn1Activate := TRUE;
   instKP8Drvs[5].btn1Mode := TRUE;
   instKP8Drvs[5].btn1ColorOn1 := 'yellow';
   instKP8Drvs[5].btn1ColorOff := 'green';
   instKP8Drvs[5].btn2Activate := TRUE;
   instKP8Drvs[5].btn2Mode := TRUE;
   instKP8Drvs[5].btn2ColorOn1 := 'yellow';
   instKP8Drvs[5].btn2ColorOff := 'green';
   instKP8Drvs[5].btn3Activate := TRUE;
   instKP8Drvs[5].btn3Mode := TRUE;
   instKP8Drvs[5].btn3ColorOn1 := 'yellow';
   instKP8Drvs[5].btn3ColorOff := 'green';
   instKP8Drvs[5].btn4ColorOn1 := 'off';
   instKP8Drvs[5].btn4ColorOn2 := 'off';
   instKP8Drvs[5].btn4ColorOff := 'off';
   instKP8Drvs[5].btn5Activate := TRUE;
   instKP8Drvs[5].btn5Mode := TRUE;
   instKP8Drvs[5].btn5ColorOn1 := 'yellow';
   instKP8Drvs[5].btn5ColorOff := 'green';
   instKP8Drvs[5].btn6Activate := TRUE;
   instKP8Drvs[5].btn6Mode := TRUE;
   instKP8Drvs[5].btn6ColorOn1 := 'yellow';
   instKP8Drvs[5].btn6ColorOff := 'green';
   instKP8Drvs[5].btn7Activate := TRUE;
   instKP8Drvs[5].btn7Mode := TRUE;
   instKP8Drvs[5].btn7ColorOn1 := 'yellow';
   instKP8Drvs[5].btn7ColorOff := 'green';
   instKP8Drvs[5].btnColorsOut := 16#00EE_0000;
   instKP8Drvs[5].i1 := 8;
   instKP8Drvs[5].i2 := 8;
   instKP8Drvs[5].btnActivateInt[1] := TRUE;
   instKP8Drvs[5].btnActivateInt[2] := TRUE;
   instKP8Drvs[5].btnActivateInt[3] := TRUE;
   instKP8Drvs[5].btnActivateInt[5] := TRUE;
   instKP8Drvs[5].btnActivateInt[6] := TRUE;
   instKP8Drvs[5].btnActivateInt[7] := TRUE;
   instKP8Drvs[5].btnClrMskOffInt[0] := 16#0000_0000;
   instKP8Drvs[5].btnClrMskOffInt[1] := 16#0002_0000;
   instKP8Drvs[5].btnClrMskOffInt[2] := 16#0004_0000;
   instKP8Drvs[5].btnClrMskOffInt[3] := 16#0008_0000;
   instKP8Drvs[5].btnClrMskOffInt[4] := 16#0000_0000;
   instKP8Drvs[5].btnClrMskOffInt[5] := 16#0020_0000;
   instKP8Drvs[5].btnClrMskOffInt[6] := 16#0040_0000;
   instKP8Drvs[5].btnClrMskOffInt[7] := 16#0080_0000;
   instKP8Drvs[5].btnClrMskOn1Int[0] := 16#0000_0000;
   instKP8Drvs[5].btnClrMskOn1Int[1] := 16#0202_0000;
   instKP8Drvs[5].btnClrMskOn1Int[2] := 16#0404_0000;
   instKP8Drvs[5].btnClrMskOn1Int[3] := 16#0808_0000;
   instKP8Drvs[5].btnClrMskOn1Int[4] := 16#0000_0000;
   instKP8Drvs[5].btnClrMskOn1Int[5] := 16#2020_0000;
   instKP8Drvs[5].btnClrMskOn1Int[6] := 16#4040_0000;
   instKP8Drvs[5].btnClrMskOn1Int[7] := 16#8080_0000;
   instKP8Drvs[5].btnClrMskOn2Int[0] := 16#0000_0000;
   instKP8Drvs[5].btnClrMskOn2Int[1] := 16#0000_0000;
   instKP8Drvs[5].btnClrMskOn2Int[2] := 16#0000_0000;
   instKP8Drvs[5].btnClrMskOn2Int[3] := 16#0000_0000;
   instKP8Drvs[5].btnClrMskOn2Int[4] := 16#0000_0000;
   instKP8Drvs[5].btnClrMskOn2Int[5] := 16#0000_0000;
   instKP8Drvs[5].btnClrMskOn2Int[6] := 16#0000_0000;
   instKP8Drvs[5].btnClrMskOn2Int[7] := 16#0000_0000;
   instKP8Drvs[5].btnClrOffInt[0] := 'off';
   instKP8Drvs[5].btnClrOffInt[1] := 'green';
   instKP8Drvs[5].btnClrOffInt[2] := 'green';
   instKP8Drvs[5].btnClrOffInt[3] := 'green';
   instKP8Drvs[5].btnClrOffInt[4] := 'off';
   instKP8Drvs[5].btnClrOffInt[5] := 'green';
   instKP8Drvs[5].btnClrOffInt[6] := 'green';
   instKP8Drvs[5].btnClrOffInt[7] := 'green';
   instKP8Drvs[5].btnClrOn1Int[0] := 'off';
   instKP8Drvs[5].btnClrOn1Int[1] := 'yellow';
   instKP8Drvs[5].btnClrOn1Int[2] := 'yellow';
   instKP8Drvs[5].btnClrOn1Int[3] := 'yellow';
   instKP8Drvs[5].btnClrOn1Int[4] := 'off';
   instKP8Drvs[5].btnClrOn1Int[5] := 'yellow';
   instKP8Drvs[5].btnClrOn1Int[6] := 'yellow';
   instKP8Drvs[5].btnClrOn1Int[7] := 'yellow';
   instKP8Drvs[5].btnClrOn2Int[0] := 'off';
   instKP8Drvs[5].btnClrOn2Int[4] := 'off';
   instKP8Drvs[5].btnColors := 16#00EE_0000;
   instKP8Drvs[5].btnModeInt[1] := TRUE;
   instKP8Drvs[5].btnModeInt[2] := TRUE;
   instKP8Drvs[5].btnModeInt[3] := TRUE;
   instKP8Drvs[5].btnModeInt[5] := TRUE;
   instKP8Drvs[5].btnModeInt[6] := TRUE;
   instKP8Drvs[5].btnModeInt[7] := TRUE;
   instKP8Drvs[6].btn0ColorOn1 := 'off';
   instKP8Drvs[6].btn0ColorOn2 := 'off';
   instKP8Drvs[6].btn0ColorOff := 'off';
   instKP8Drvs[6].btn1Activate := TRUE;
   instKP8Drvs[6].btn1Mode := TRUE;
   instKP8Drvs[6].btn1ColorOn1 := 'yellow';
   instKP8Drvs[6].btn1ColorOff := 'green';
   instKP8Drvs[6].btn2Activate := TRUE;
   instKP8Drvs[6].btn2Mode := TRUE;
   instKP8Drvs[6].btn2ColorOn1 := 'yellow';
   instKP8Drvs[6].btn2ColorOff := 'green';
   instKP8Drvs[6].btn3Activate := TRUE;
   instKP8Drvs[6].btn3Mode := TRUE;
   instKP8Drvs[6].btn3ColorOn1 := 'yellow';
   instKP8Drvs[6].btn3ColorOff := 'green';
   instKP8Drvs[6].btn4ColorOn1 := 'off';
   instKP8Drvs[6].btn4ColorOn2 := 'off';
   instKP8Drvs[6].btn4ColorOff := 'off';
   instKP8Drvs[6].btn5Activate := TRUE;
   instKP8Drvs[6].btn5Mode := TRUE;
   instKP8Drvs[6].btn5ColorOn1 := 'yellow';
   instKP8Drvs[6].btn5ColorOff := 'green';
   instKP8Drvs[6].btn6Activate := TRUE;
   instKP8Drvs[6].btn6Mode := TRUE;
   instKP8Drvs[6].btn6ColorOn1 := 'yellow';
   instKP8Drvs[6].btn6ColorOff := 'green';
   instKP8Drvs[6].btn7Activate := TRUE;
   instKP8Drvs[6].btn7Mode := TRUE;
   instKP8Drvs[6].btn7ColorOn1 := 'yellow';
   instKP8Drvs[6].btn7ColorOff := 'green';
   instKP8Drvs[6].btnColorsOut := 16#00EE_0000;
   instKP8Drvs[6].i1 := 8;
   instKP8Drvs[6].i2 := 8;
   instKP8Drvs[6].btnActivateInt[1] := TRUE;
   instKP8Drvs[6].btnActivateInt[2] := TRUE;
   instKP8Drvs[6].btnActivateInt[3] := TRUE;
   instKP8Drvs[6].btnActivateInt[5] := TRUE;
   instKP8Drvs[6].btnActivateInt[6] := TRUE;
   instKP8Drvs[6].btnActivateInt[7] := TRUE;
   instKP8Drvs[6].btnClrMskOffInt[0] := 16#0000_0000;
   instKP8Drvs[6].btnClrMskOffInt[1] := 16#0002_0000;
   instKP8Drvs[6].btnClrMskOffInt[2] := 16#0004_0000;
   instKP8Drvs[6].btnClrMskOffInt[3] := 16#0008_0000;
   instKP8Drvs[6].btnClrMskOffInt[4] := 16#0000_0000;
   instKP8Drvs[6].btnClrMskOffInt[5] := 16#0020_0000;
   instKP8Drvs[6].btnClrMskOffInt[6] := 16#0040_0000;
   instKP8Drvs[6].btnClrMskOffInt[7] := 16#0080_0000;
   instKP8Drvs[6].btnClrMskOn1Int[0] := 16#0000_0000;
   instKP8Drvs[6].btnClrMskOn1Int[1] := 16#0202_0000;
   instKP8Drvs[6].btnClrMskOn1Int[2] := 16#0404_0000;
   instKP8Drvs[6].btnClrMskOn1Int[3] := 16#0808_0000;
   instKP8Drvs[6].btnClrMskOn1Int[4] := 16#0000_0000;
   instKP8Drvs[6].btnClrMskOn1Int[5] := 16#2020_0000;
   instKP8Drvs[6].btnClrMskOn1Int[6] := 16#4040_0000;
   instKP8Drvs[6].btnClrMskOn1Int[7] := 16#8080_0000;
   instKP8Drvs[6].btnClrMskOn2Int[0] := 16#0000_0000;
   instKP8Drvs[6].btnClrMskOn2Int[1] := 16#0000_0000;
   instKP8Drvs[6].btnClrMskOn2Int[2] := 16#0000_0000;
   instKP8Drvs[6].btnClrMskOn2Int[3] := 16#0000_0000;
   instKP8Drvs[6].btnClrMskOn2Int[4] := 16#0000_0000;
   instKP8Drvs[6].btnClrMskOn2Int[5] := 16#0000_0000;
   instKP8Drvs[6].btnClrMskOn2Int[6] := 16#0000_0000;
   instKP8Drvs[6].btnClrMskOn2Int[7] := 16#0000_0000;
   instKP8Drvs[6].btnClrOffInt[0] := 'off';
   instKP8Drvs[6].btnClrOffInt[1] := 'green';
   instKP8Drvs[6].btnClrOffInt[2] := 'green';
   instKP8Drvs[6].btnClrOffInt[3] := 'green';
   instKP8Drvs[6].btnClrOffInt[4] := 'off';
   instKP8Drvs[6].btnClrOffInt[5] := 'green';
   instKP8Drvs[6].btnClrOffInt[6] := 'green';
   instKP8Drvs[6].btnClrOffInt[7] := 'green';
   instKP8Drvs[6].btnClrOn1Int[0] := 'off';
   instKP8Drvs[6].btnClrOn1Int[1] := 'yellow';
   instKP8Drvs[6].btnClrOn1Int[2] := 'yellow';
   instKP8Drvs[6].btnClrOn1Int[3] := 'yellow';
   instKP8Drvs[6].btnClrOn1Int[4] := 'off';
   instKP8Drvs[6].btnClrOn1Int[5] := 'yellow';
   instKP8Drvs[6].btnClrOn1Int[6] := 'yellow';
   instKP8Drvs[6].btnClrOn1Int[7] := 'yellow';
   instKP8Drvs[6].btnClrOn2Int[0] := 'off';
   instKP8Drvs[6].btnClrOn2Int[4] := 'off';
   instKP8Drvs[6].btnColors := 16#00EE_0000;
   instKP8Drvs[6].btnModeInt[1] := TRUE;
   instKP8Drvs[6].btnModeInt[2] := TRUE;
   instKP8Drvs[6].btnModeInt[3] := TRUE;
   instKP8Drvs[6].btnModeInt[5] := TRUE;
   instKP8Drvs[6].btnModeInt[6] := TRUE;
   instKP8Drvs[6].btnModeInt[7] := TRUE;
   instKP8Drvs[7].btn0ColorOn1 := 'off';
   instKP8Drvs[7].btn0ColorOn2 := 'off';
   instKP8Drvs[7].btn0ColorOff := 'off';
   instKP8Drvs[7].btn1ColorOn1 := 'off';
   instKP8Drvs[7].btn1ColorOn2 := 'off';
   instKP8Drvs[7].btn1ColorOff := 'off';
   instKP8Drvs[7].btn2ColorOn1 := 'off';
   instKP8Drvs[7].btn2ColorOn2 := 'off';
   instKP8Drvs[7].btn2ColorOff := 'off';
   instKP8Drvs[7].btn3Activate := TRUE;
   instKP8Drvs[7].btn3Mode := TRUE;
   instKP8Drvs[7].btn3ColorOn1 := 'yellow';
   instKP8Drvs[7].btn3ColorOff := 'green';
   instKP8Drvs[7].btn4ColorOn1 := 'off';
   instKP8Drvs[7].btn4ColorOn2 := 'off';
   instKP8Drvs[7].btn4ColorOff := 'off';
   instKP8Drvs[7].btn5ColorOn1 := 'off';
   instKP8Drvs[7].btn5ColorOn2 := 'off';
   instKP8Drvs[7].btn5ColorOff := 'off';
   instKP8Drvs[7].btn6Activate := TRUE;
   instKP8Drvs[7].btn6Mode := TRUE;
   instKP8Drvs[7].btn6ColorOn1 := 'yellow';
   instKP8Drvs[7].btn6ColorOff := 'green';
   instKP8Drvs[7].btn7Activate := TRUE;
   instKP8Drvs[7].btn7Mode := TRUE;
   instKP8Drvs[7].btn7ColorOn1 := 'yellow';
   instKP8Drvs[7].btn7ColorOff := 'green';
   instKP8Drvs[7].btnColorsOut := 16#00C8_0000;
   instKP8Drvs[7].i1 := 8;
   instKP8Drvs[7].i2 := 8;
   instKP8Drvs[7].btnActivateInt[3] := TRUE;
   instKP8Drvs[7].btnActivateInt[6] := TRUE;
   instKP8Drvs[7].btnActivateInt[7] := TRUE;
   instKP8Drvs[7].btnClrMskOffInt[0] := 16#0000_0000;
   instKP8Drvs[7].btnClrMskOffInt[1] := 16#0000_0000;
   instKP8Drvs[7].btnClrMskOffInt[2] := 16#0000_0000;
   instKP8Drvs[7].btnClrMskOffInt[3] := 16#0008_0000;
   instKP8Drvs[7].btnClrMskOffInt[4] := 16#0000_0000;
   instKP8Drvs[7].btnClrMskOffInt[5] := 16#0000_0000;
   instKP8Drvs[7].btnClrMskOffInt[6] := 16#0040_0000;
   instKP8Drvs[7].btnClrMskOffInt[7] := 16#0080_0000;
   instKP8Drvs[7].btnClrMskOn1Int[0] := 16#0000_0000;
   instKP8Drvs[7].btnClrMskOn1Int[1] := 16#0000_0000;
   instKP8Drvs[7].btnClrMskOn1Int[2] := 16#0000_0000;
   instKP8Drvs[7].btnClrMskOn1Int[3] := 16#0808_0000;
   instKP8Drvs[7].btnClrMskOn1Int[4] := 16#0000_0000;
   instKP8Drvs[7].btnClrMskOn1Int[5] := 16#0000_0000;
   instKP8Drvs[7].btnClrMskOn1Int[6] := 16#4040_0000;
   instKP8Drvs[7].btnClrMskOn1Int[7] := 16#8080_0000;
   instKP8Drvs[7].btnClrMskOn2Int[0] := 16#0000_0000;
   instKP8Drvs[7].btnClrMskOn2Int[1] := 16#0000_0000;
   instKP8Drvs[7].btnClrMskOn2Int[2] := 16#0000_0000;
   instKP8Drvs[7].btnClrMskOn2Int[3] := 16#0000_0000;
   instKP8Drvs[7].btnClrMskOn2Int[4] := 16#0000_0000;
   instKP8Drvs[7].btnClrMskOn2Int[5] := 16#0000_0000;
   instKP8Drvs[7].btnClrMskOn2Int[6] := 16#0000_0000;
   instKP8Drvs[7].btnClrMskOn2Int[7] := 16#0000_0000;
   instKP8Drvs[7].btnClrOffInt[0] := 'off';
   instKP8Drvs[7].btnClrOffInt[1] := 'off';
   instKP8Drvs[7].btnClrOffInt[2] := 'off';
   instKP8Drvs[7].btnClrOffInt[3] := 'green';
   instKP8Drvs[7].btnClrOffInt[4] := 'off';
   instKP8Drvs[7].btnClrOffInt[5] := 'off';
   instKP8Drvs[7].btnClrOffInt[6] := 'green';
   instKP8Drvs[7].btnClrOffInt[7] := 'green';
   instKP8Drvs[7].btnClrOn1Int[0] := 'off';
   instKP8Drvs[7].btnClrOn1Int[1] := 'off';
   instKP8Drvs[7].btnClrOn1Int[2] := 'off';
   instKP8Drvs[7].btnClrOn1Int[3] := 'yellow';
   instKP8Drvs[7].btnClrOn1Int[4] := 'off';
   instKP8Drvs[7].btnClrOn1Int[5] := 'off';
   instKP8Drvs[7].btnClrOn1Int[6] := 'yellow';
   instKP8Drvs[7].btnClrOn1Int[7] := 'yellow';
   instKP8Drvs[7].btnClrOn2Int[0] := 'off';
   instKP8Drvs[7].btnClrOn2Int[1] := 'off';
   instKP8Drvs[7].btnClrOn2Int[2] := 'off';
   instKP8Drvs[7].btnClrOn2Int[4] := 'off';
   instKP8Drvs[7].btnClrOn2Int[5] := 'off';
   instKP8Drvs[7].btnColors := 16#00C8_0000;
   instKP8Drvs[7].btnModeInt[3] := TRUE;
   instKP8Drvs[7].btnModeInt[6] := TRUE;
   instKP8Drvs[7].btnModeInt[7] := TRUE;
   instKP8Drvs[8].btn0ColorOn1 := 'off';
   instKP8Drvs[8].btn0ColorOn2 := 'off';
   instKP8Drvs[8].btn0ColorOff := 'off';
   instKP8Drvs[8].btn1ColorOn1 := 'off';
   instKP8Drvs[8].btn1ColorOn2 := 'off';
   instKP8Drvs[8].btn1ColorOff := 'off';
   instKP8Drvs[8].btn2ColorOn1 := 'off';
   instKP8Drvs[8].btn2ColorOn2 := 'off';
   instKP8Drvs[8].btn2ColorOff := 'off';
   instKP8Drvs[8].btn3Activate := TRUE;
   instKP8Drvs[8].btn3Mode := TRUE;
   instKP8Drvs[8].btn3ColorOn1 := 'yellow';
   instKP8Drvs[8].btn3ColorOff := 'green';
   instKP8Drvs[8].btn4ColorOn1 := 'off';
   instKP8Drvs[8].btn4ColorOn2 := 'off';
   instKP8Drvs[8].btn4ColorOff := 'off';
   instKP8Drvs[8].btn5ColorOn1 := 'off';
   instKP8Drvs[8].btn5ColorOn2 := 'off';
   instKP8Drvs[8].btn5ColorOff := 'off';
   instKP8Drvs[8].btn6Activate := TRUE;
   instKP8Drvs[8].btn6Mode := TRUE;
   instKP8Drvs[8].btn6ColorOn1 := 'yellow';
   instKP8Drvs[8].btn6ColorOff := 'green';
   instKP8Drvs[8].btn7Activate := TRUE;
   instKP8Drvs[8].btn7Mode := TRUE;
   instKP8Drvs[8].btn7ColorOn1 := 'yellow';
   instKP8Drvs[8].btn7ColorOff := 'green';
   instKP8Drvs[8].btnColorsOut := 16#00C8_0000;
   instKP8Drvs[8].i1 := 8;
   instKP8Drvs[8].i2 := 8;
   instKP8Drvs[8].btnActivateInt[3] := TRUE;
   instKP8Drvs[8].btnActivateInt[6] := TRUE;
   instKP8Drvs[8].btnActivateInt[7] := TRUE;
   instKP8Drvs[8].btnClrMskOffInt[0] := 16#0000_0000;
   instKP8Drvs[8].btnClrMskOffInt[1] := 16#0000_0000;
   instKP8Drvs[8].btnClrMskOffInt[2] := 16#0000_0000;
   instKP8Drvs[8].btnClrMskOffInt[3] := 16#0008_0000;
   instKP8Drvs[8].btnClrMskOffInt[4] := 16#0000_0000;
   instKP8Drvs[8].btnClrMskOffInt[5] := 16#0000_0000;
   instKP8Drvs[8].btnClrMskOffInt[6] := 16#0040_0000;
   instKP8Drvs[8].btnClrMskOffInt[7] := 16#0080_0000;
   instKP8Drvs[8].btnClrMskOn1Int[0] := 16#0000_0000;
   instKP8Drvs[8].btnClrMskOn1Int[1] := 16#0000_0000;
   instKP8Drvs[8].btnClrMskOn1Int[2] := 16#0000_0000;
   instKP8Drvs[8].btnClrMskOn1Int[3] := 16#0808_0000;
   instKP8Drvs[8].btnClrMskOn1Int[4] := 16#0000_0000;
   instKP8Drvs[8].btnClrMskOn1Int[5] := 16#0000_0000;
   instKP8Drvs[8].btnClrMskOn1Int[6] := 16#4040_0000;
   instKP8Drvs[8].btnClrMskOn1Int[7] := 16#8080_0000;
   instKP8Drvs[8].btnClrMskOn2Int[0] := 16#0000_0000;
   instKP8Drvs[8].btnClrMskOn2Int[1] := 16#0000_0000;
   instKP8Drvs[8].btnClrMskOn2Int[2] := 16#0000_0000;
   instKP8Drvs[8].btnClrMskOn2Int[3] := 16#0000_0000;
   instKP8Drvs[8].btnClrMskOn2Int[4] := 16#0000_0000;
   instKP8Drvs[8].btnClrMskOn2Int[5] := 16#0000_0000;
   instKP8Drvs[8].btnClrMskOn2Int[6] := 16#0000_0000;
   instKP8Drvs[8].btnClrMskOn2Int[7] := 16#0000_0000;
   instKP8Drvs[8].btnClrOffInt[0] := 'off';
   instKP8Drvs[8].btnClrOffInt[1] := 'off';
   instKP8Drvs[8].btnClrOffInt[2] := 'off';
   instKP8Drvs[8].btnClrOffInt[3] := 'green';
   instKP8Drvs[8].btnClrOffInt[4] := 'off';
   instKP8Drvs[8].btnClrOffInt[5] := 'off';
   instKP8Drvs[8].btnClrOffInt[6] := 'green';
   instKP8Drvs[8].btnClrOffInt[7] := 'green';
   instKP8Drvs[8].btnClrOn1Int[0] := 'off';
   instKP8Drvs[8].btnClrOn1Int[1] := 'off';
   instKP8Drvs[8].btnClrOn1Int[2] := 'off';
   instKP8Drvs[8].btnClrOn1Int[3] := 'yellow';
   instKP8Drvs[8].btnClrOn1Int[4] := 'off';
   instKP8Drvs[8].btnClrOn1Int[5] := 'off';
   instKP8Drvs[8].btnClrOn1Int[6] := 'yellow';
   instKP8Drvs[8].btnClrOn1Int[7] := 'yellow';
   instKP8Drvs[8].btnClrOn2Int[0] := 'off';
   instKP8Drvs[8].btnClrOn2Int[1] := 'off';
   instKP8Drvs[8].btnClrOn2Int[2] := 'off';
   instKP8Drvs[8].btnClrOn2Int[4] := 'off';
   instKP8Drvs[8].btnClrOn2Int[5] := 'off';
   instKP8Drvs[8].btnColors := 16#00C8_0000;
   instKP8Drvs[8].btnModeInt[3] := TRUE;
   instKP8Drvs[8].btnModeInt[6] := TRUE;
   instKP8Drvs[8].btnModeInt[7] := TRUE;
   instKP8Drvs[9].btn0ColorOn1 := 'off';
   instKP8Drvs[9].btn0ColorOn2 := 'off';
   instKP8Drvs[9].btn0ColorOff := 'off';
   instKP8Drvs[9].btn1ColorOn1 := 'off';
   instKP8Drvs[9].btn1ColorOn2 := 'off';
   instKP8Drvs[9].btn1ColorOff := 'off';
   instKP8Drvs[9].btn2ColorOn1 := 'off';
   instKP8Drvs[9].btn2ColorOn2 := 'off';
   instKP8Drvs[9].btn2ColorOff := 'off';
   instKP8Drvs[9].btn3Activate := TRUE;
   instKP8Drvs[9].btn3Mode := TRUE;
   instKP8Drvs[9].btn3ColorOn1 := 'yellow';
   instKP8Drvs[9].btn3ColorOff := 'green';
   instKP8Drvs[9].btn4ColorOn1 := 'off';
   instKP8Drvs[9].btn4ColorOn2 := 'off';
   instKP8Drvs[9].btn4ColorOff := 'off';
   instKP8Drvs[9].btn5ColorOn1 := 'off';
   instKP8Drvs[9].btn5ColorOn2 := 'off';
   instKP8Drvs[9].btn5ColorOff := 'off';
   instKP8Drvs[9].btn6ColorOn1 := 'off';
   instKP8Drvs[9].btn6ColorOn2 := 'off';
   instKP8Drvs[9].btn6ColorOff := 'off';
   instKP8Drvs[9].btn7Activate := TRUE;
   instKP8Drvs[9].btn7Mode := TRUE;
   instKP8Drvs[9].btn7ColorOn1 := 'yellow';
   instKP8Drvs[9].btn7ColorOff := 'green';
   instKP8Drvs[9].btnColorsOut := 16#0088_0000;
   instKP8Drvs[9].i1 := 8;
   instKP8Drvs[9].i2 := 8;
   instKP8Drvs[9].btnActivateInt[3] := TRUE;
   instKP8Drvs[9].btnActivateInt[7] := TRUE;
   instKP8Drvs[9].btnClrMskOffInt[0] := 16#0000_0000;
   instKP8Drvs[9].btnClrMskOffInt[1] := 16#0000_0000;
   instKP8Drvs[9].btnClrMskOffInt[2] := 16#0000_0000;
   instKP8Drvs[9].btnClrMskOffInt[3] := 16#0008_0000;
   instKP8Drvs[9].btnClrMskOffInt[4] := 16#0000_0000;
   instKP8Drvs[9].btnClrMskOffInt[5] := 16#0000_0000;
   instKP8Drvs[9].btnClrMskOffInt[6] := 16#0000_0000;
   instKP8Drvs[9].btnClrMskOffInt[7] := 16#0080_0000;
   instKP8Drvs[9].btnClrMskOn1Int[0] := 16#0000_0000;
   instKP8Drvs[9].btnClrMskOn1Int[1] := 16#0000_0000;
   instKP8Drvs[9].btnClrMskOn1Int[2] := 16#0000_0000;
   instKP8Drvs[9].btnClrMskOn1Int[3] := 16#0808_0000;
   instKP8Drvs[9].btnClrMskOn1Int[4] := 16#0000_0000;
   instKP8Drvs[9].btnClrMskOn1Int[5] := 16#0000_0000;
   instKP8Drvs[9].btnClrMskOn1Int[6] := 16#0000_0000;
   instKP8Drvs[9].btnClrMskOn1Int[7] := 16#8080_0000;
   instKP8Drvs[9].btnClrMskOn2Int[0] := 16#0000_0000;
   instKP8Drvs[9].btnClrMskOn2Int[1] := 16#0000_0000;
   instKP8Drvs[9].btnClrMskOn2Int[2] := 16#0000_0000;
   instKP8Drvs[9].btnClrMskOn2Int[3] := 16#0000_0000;
   instKP8Drvs[9].btnClrMskOn2Int[4] := 16#0000_0000;
   instKP8Drvs[9].btnClrMskOn2Int[5] := 16#0000_0000;
   instKP8Drvs[9].btnClrMskOn2Int[6] := 16#0000_0000;
   instKP8Drvs[9].btnClrMskOn2Int[7] := 16#0000_0000;
   instKP8Drvs[9].btnClrOffInt[0] := 'off';
   instKP8Drvs[9].btnClrOffInt[1] := 'off';
   instKP8Drvs[9].btnClrOffInt[2] := 'off';
   instKP8Drvs[9].btnClrOffInt[3] := 'green';
   instKP8Drvs[9].btnClrOffInt[4] := 'off';
   instKP8Drvs[9].btnClrOffInt[5] := 'off';
   instKP8Drvs[9].btnClrOffInt[6] := 'off';
   instKP8Drvs[9].btnClrOffInt[7] := 'green';
   instKP8Drvs[9].btnClrOn1Int[0] := 'off';
   instKP8Drvs[9].btnClrOn1Int[1] := 'off';
   instKP8Drvs[9].btnClrOn1Int[2] := 'off';
   instKP8Drvs[9].btnClrOn1Int[3] := 'yellow';
   instKP8Drvs[9].btnClrOn1Int[4] := 'off';
   instKP8Drvs[9].btnClrOn1Int[5] := 'off';
   instKP8Drvs[9].btnClrOn1Int[6] := 'off';
   instKP8Drvs[9].btnClrOn1Int[7] := 'yellow';
   instKP8Drvs[9].btnClrOn2Int[0] := 'off';
   instKP8Drvs[9].btnClrOn2Int[1] := 'off';
   instKP8Drvs[9].btnClrOn2Int[2] := 'off';
   instKP8Drvs[9].btnClrOn2Int[4] := 'off';
   instKP8Drvs[9].btnClrOn2Int[5] := 'off';
   instKP8Drvs[9].btnClrOn2Int[6] := 'off';
   instKP8Drvs[9].btnColors := 16#0088_0000;
   instKP8Drvs[9].btnModeInt[3] := TRUE;
   instKP8Drvs[9].btnModeInt[7] := TRUE;
   instKP8Drvs[10].btn0ColorOn1 := 'off';
   instKP8Drvs[10].btn0ColorOn2 := 'off';
   instKP8Drvs[10].btn0ColorOff := 'off';
   instKP8Drvs[10].btn1ColorOn1 := 'off';
   instKP8Drvs[10].btn1ColorOn2 := 'off';
   instKP8Drvs[10].btn1ColorOff := 'off';
   instKP8Drvs[10].btn2ColorOn1 := 'off';
   instKP8Drvs[10].btn2ColorOn2 := 'off';
   instKP8Drvs[10].btn2ColorOff := 'off';
   instKP8Drvs[10].btn3Activate := TRUE;
   instKP8Drvs[10].btn3Mode := TRUE;
   instKP8Drvs[10].btn3ColorOn1 := 'yellow';
   instKP8Drvs[10].btn3ColorOff := 'green';
   instKP8Drvs[10].btn4ColorOn1 := 'off';
   instKP8Drvs[10].btn4ColorOn2 := 'off';
   instKP8Drvs[10].btn4ColorOff := 'off';
   instKP8Drvs[10].btn5ColorOn1 := 'off';
   instKP8Drvs[10].btn5ColorOn2 := 'off';
   instKP8Drvs[10].btn5ColorOff := 'off';
   instKP8Drvs[10].btn6Activate := TRUE;
   instKP8Drvs[10].btn6Mode := TRUE;
   instKP8Drvs[10].btn6ColorOn1 := 'yellow';
   instKP8Drvs[10].btn6ColorOff := 'green';
   instKP8Drvs[10].btn7Activate := TRUE;
   instKP8Drvs[10].btn7Mode := TRUE;
   instKP8Drvs[10].btn7ColorOn1 := 'yellow';
   instKP8Drvs[10].btn7ColorOff := 'green';
   instKP8Drvs[10].btnColorsOut := 16#00C8_0000;
   instKP8Drvs[10].i1 := 8;
   instKP8Drvs[10].i2 := 8;
   instKP8Drvs[10].btnActivateInt[3] := TRUE;
   instKP8Drvs[10].btnActivateInt[6] := TRUE;
   instKP8Drvs[10].btnActivateInt[7] := TRUE;
   instKP8Drvs[10].btnClrMskOffInt[0] := 16#0000_0000;
   instKP8Drvs[10].btnClrMskOffInt[1] := 16#0000_0000;
   instKP8Drvs[10].btnClrMskOffInt[2] := 16#0000_0000;
   instKP8Drvs[10].btnClrMskOffInt[3] := 16#0008_0000;
   instKP8Drvs[10].btnClrMskOffInt[4] := 16#0000_0000;
   instKP8Drvs[10].btnClrMskOffInt[5] := 16#0000_0000;
   instKP8Drvs[10].btnClrMskOffInt[6] := 16#0040_0000;
   instKP8Drvs[10].btnClrMskOffInt[7] := 16#0080_0000;
   instKP8Drvs[10].btnClrMskOn1Int[0] := 16#0000_0000;
   instKP8Drvs[10].btnClrMskOn1Int[1] := 16#0000_0000;
   instKP8Drvs[10].btnClrMskOn1Int[2] := 16#0000_0000;
   instKP8Drvs[10].btnClrMskOn1Int[3] := 16#0808_0000;
   instKP8Drvs[10].btnClrMskOn1Int[4] := 16#0000_0000;
   instKP8Drvs[10].btnClrMskOn1Int[5] := 16#0000_0000;
   instKP8Drvs[10].btnClrMskOn1Int[6] := 16#4040_0000;
   instKP8Drvs[10].btnClrMskOn1Int[7] := 16#8080_0000;
   instKP8Drvs[10].btnClrMskOn2Int[0] := 16#0000_0000;
   instKP8Drvs[10].btnClrMskOn2Int[1] := 16#0000_0000;
   instKP8Drvs[10].btnClrMskOn2Int[2] := 16#0000_0000;
   instKP8Drvs[10].btnClrMskOn2Int[3] := 16#0000_0000;
   instKP8Drvs[10].btnClrMskOn2Int[4] := 16#0000_0000;
   instKP8Drvs[10].btnClrMskOn2Int[5] := 16#0000_0000;
   instKP8Drvs[10].btnClrMskOn2Int[6] := 16#0000_0000;
   instKP8Drvs[10].btnClrMskOn2Int[7] := 16#0000_0000;
   instKP8Drvs[10].btnClrOffInt[0] := 'off';
   instKP8Drvs[10].btnClrOffInt[1] := 'off';
   instKP8Drvs[10].btnClrOffInt[2] := 'off';
   instKP8Drvs[10].btnClrOffInt[3] := 'green';
   instKP8Drvs[10].btnClrOffInt[4] := 'off';
   instKP8Drvs[10].btnClrOffInt[5] := 'off';
   instKP8Drvs[10].btnClrOffInt[6] := 'green';
   instKP8Drvs[10].btnClrOffInt[7] := 'green';
   instKP8Drvs[10].btnClrOn1Int[0] := 'off';
   instKP8Drvs[10].btnClrOn1Int[1] := 'off';
   instKP8Drvs[10].btnClrOn1Int[2] := 'off';
   instKP8Drvs[10].btnClrOn1Int[3] := 'yellow';
   instKP8Drvs[10].btnClrOn1Int[4] := 'off';
   instKP8Drvs[10].btnClrOn1Int[5] := 'off';
   instKP8Drvs[10].btnClrOn1Int[6] := 'yellow';
   instKP8Drvs[10].btnClrOn1Int[7] := 'yellow';
   instKP8Drvs[10].btnClrOn2Int[0] := 'off';
   instKP8Drvs[10].btnClrOn2Int[1] := 'off';
   instKP8Drvs[10].btnClrOn2Int[2] := 'off';
   instKP8Drvs[10].btnClrOn2Int[4] := 'off';
   instKP8Drvs[10].btnClrOn2Int[5] := 'off';
   instKP8Drvs[10].btnColors := 16#00C8_0000;
   instKP8Drvs[10].btnModeInt[3] := TRUE;
   instKP8Drvs[10].btnModeInt[6] := TRUE;
   instKP8Drvs[10].btnModeInt[7] := TRUE;
   instKP8Drvs[11].btn0ColorOn1 := 'off';
   instKP8Drvs[11].btn0ColorOn2 := 'off';
   instKP8Drvs[11].btn0ColorOff := 'off';
   instKP8Drvs[11].btn1ColorOn1 := 'off';
   instKP8Drvs[11].btn1ColorOn2 := 'off';
   instKP8Drvs[11].btn1ColorOff := 'off';
   instKP8Drvs[11].btn2ColorOn1 := 'off';
   instKP8Drvs[11].btn2ColorOn2 := 'off';
   instKP8Drvs[11].btn2ColorOff := 'off';
   instKP8Drvs[11].btn3Activate := TRUE;
   instKP8Drvs[11].btn3Mode := TRUE;
   instKP8Drvs[11].btn3ColorOn1 := 'yellow';
   instKP8Drvs[11].btn3ColorOff := 'green';
   instKP8Drvs[11].btn4ColorOn1 := 'off';
   instKP8Drvs[11].btn4ColorOn2 := 'off';
   instKP8Drvs[11].btn4ColorOff := 'off';
   instKP8Drvs[11].btn5ColorOn1 := 'off';
   instKP8Drvs[11].btn5ColorOn2 := 'off';
   instKP8Drvs[11].btn5ColorOff := 'off';
   instKP8Drvs[11].btn6Activate := TRUE;
   instKP8Drvs[11].btn6Mode := TRUE;
   instKP8Drvs[11].btn6ColorOn1 := 'yellow';
   instKP8Drvs[11].btn6ColorOff := 'green';
   instKP8Drvs[11].btn7Activate := TRUE;
   instKP8Drvs[11].btn7Mode := TRUE;
   instKP8Drvs[11].btn7ColorOn1 := 'yellow';
   instKP8Drvs[11].btn7ColorOff := 'green';
   instKP8Drvs[11].btnColorsOut := 16#00C8_0000;
   instKP8Drvs[11].i1 := 8;
   instKP8Drvs[11].i2 := 8;
   instKP8Drvs[11].btnActivateInt[3] := TRUE;
   instKP8Drvs[11].btnActivateInt[6] := TRUE;
   instKP8Drvs[11].btnActivateInt[7] := TRUE;
   instKP8Drvs[11].btnClrMskOffInt[0] := 16#0000_0000;
   instKP8Drvs[11].btnClrMskOffInt[1] := 16#0000_0000;
   instKP8Drvs[11].btnClrMskOffInt[2] := 16#0000_0000;
   instKP8Drvs[11].btnClrMskOffInt[3] := 16#0008_0000;
   instKP8Drvs[11].btnClrMskOffInt[4] := 16#0000_0000;
   instKP8Drvs[11].btnClrMskOffInt[5] := 16#0000_0000;
   instKP8Drvs[11].btnClrMskOffInt[6] := 16#0040_0000;
   instKP8Drvs[11].btnClrMskOffInt[7] := 16#0080_0000;
   instKP8Drvs[11].btnClrMskOn1Int[0] := 16#0000_0000;
   instKP8Drvs[11].btnClrMskOn1Int[1] := 16#0000_0000;
   instKP8Drvs[11].btnClrMskOn1Int[2] := 16#0000_0000;
   instKP8Drvs[11].btnClrMskOn1Int[3] := 16#0808_0000;
   instKP8Drvs[11].btnClrMskOn1Int[4] := 16#0000_0000;
   instKP8Drvs[11].btnClrMskOn1Int[5] := 16#0000_0000;
   instKP8Drvs[11].btnClrMskOn1Int[6] := 16#4040_0000;
   instKP8Drvs[11].btnClrMskOn1Int[7] := 16#8080_0000;
   instKP8Drvs[11].btnClrMskOn2Int[0] := 16#0000_0000;
   instKP8Drvs[11].btnClrMskOn2Int[1] := 16#0000_0000;
   instKP8Drvs[11].btnClrMskOn2Int[2] := 16#0000_0000;
   instKP8Drvs[11].btnClrMskOn2Int[3] := 16#0000_0000;
   instKP8Drvs[11].btnClrMskOn2Int[4] := 16#0000_0000;
   instKP8Drvs[11].btnClrMskOn2Int[5] := 16#0000_0000;
   instKP8Drvs[11].btnClrMskOn2Int[6] := 16#0000_0000;
   instKP8Drvs[11].btnClrMskOn2Int[7] := 16#0000_0000;
   instKP8Drvs[11].btnClrOffInt[0] := 'off';
   instKP8Drvs[11].btnClrOffInt[1] := 'off';
   instKP8Drvs[11].btnClrOffInt[2] := 'off';
   instKP8Drvs[11].btnClrOffInt[3] := 'green';
   instKP8Drvs[11].btnClrOffInt[4] := 'off';
   instKP8Drvs[11].btnClrOffInt[5] := 'off';
   instKP8Drvs[11].btnClrOffInt[6] := 'green';
   instKP8Drvs[11].btnClrOffInt[7] := 'green';
   instKP8Drvs[11].btnClrOn1Int[0] := 'off';
   instKP8Drvs[11].btnClrOn1Int[1] := 'off';
   instKP8Drvs[11].btnClrOn1Int[2] := 'off';
   instKP8Drvs[11].btnClrOn1Int[3] := 'yellow';
   instKP8Drvs[11].btnClrOn1Int[4] := 'off';
   instKP8Drvs[11].btnClrOn1Int[5] := 'off';
   instKP8Drvs[11].btnClrOn1Int[6] := 'yellow';
   instKP8Drvs[11].btnClrOn1Int[7] := 'yellow';
   instKP8Drvs[11].btnClrOn2Int[0] := 'off';
   instKP8Drvs[11].btnClrOn2Int[1] := 'off';
   instKP8Drvs[11].btnClrOn2Int[2] := 'off';
   instKP8Drvs[11].btnClrOn2Int[4] := 'off';
   instKP8Drvs[11].btnClrOn2Int[5] := 'off';
   instKP8Drvs[11].btnColors := 16#00C8_0000;
   instKP8Drvs[11].btnModeInt[3] := TRUE;
   instKP8Drvs[11].btnModeInt[6] := TRUE;
   instKP8Drvs[11].btnModeInt[7] := TRUE;
   instKP8Drvs[12].btn0ColorOn1 := 'off';
   instKP8Drvs[12].btn0ColorOn2 := 'off';
   instKP8Drvs[12].btn0ColorOff := 'off';
   instKP8Drvs[12].btn1Activate := TRUE;
   instKP8Drvs[12].btn1Mode := TRUE;
   instKP8Drvs[12].btn1ColorOn1 := 'yellow';
   instKP8Drvs[12].btn1ColorOff := 'green';
   instKP8Drvs[12].btn2Activate := TRUE;
   instKP8Drvs[12].btn2Mode := TRUE;
   instKP8Drvs[12].btn2ColorOn1 := 'yellow';
   instKP8Drvs[12].btn2ColorOff := 'green';
   instKP8Drvs[12].btn3Activate := TRUE;
   instKP8Drvs[12].btn3Mode := TRUE;
   instKP8Drvs[12].btn3ColorOn1 := 'yellow';
   instKP8Drvs[12].btn3ColorOff := 'green';
   instKP8Drvs[12].btn4ColorOn1 := 'off';
   instKP8Drvs[12].btn4ColorOn2 := 'off';
   instKP8Drvs[12].btn4ColorOff := 'off';
   instKP8Drvs[12].btn5Activate := TRUE;
   instKP8Drvs[12].btn5Mode := TRUE;
   instKP8Drvs[12].btn5ColorOn1 := 'yellow';
   instKP8Drvs[12].btn5ColorOff := 'green';
   instKP8Drvs[12].btn6Activate := TRUE;
   instKP8Drvs[12].btn6Mode := TRUE;
   instKP8Drvs[12].btn6ColorOn1 := 'yellow';
   instKP8Drvs[12].btn6ColorOff := 'green';
   instKP8Drvs[12].btn7Activate := TRUE;
   instKP8Drvs[12].btn7Mode := TRUE;
   instKP8Drvs[12].btn7ColorOn1 := 'yellow';
   instKP8Drvs[12].btn7ColorOff := 'green';
   instKP8Drvs[12].btnColorsOut := 16#00EE_0000;
   instKP8Drvs[12].i1 := 8;
   instKP8Drvs[12].i2 := 8;
   instKP8Drvs[12].btnActivateInt[1] := TRUE;
   instKP8Drvs[12].btnActivateInt[2] := TRUE;
   instKP8Drvs[12].btnActivateInt[3] := TRUE;
   instKP8Drvs[12].btnActivateInt[5] := TRUE;
   instKP8Drvs[12].btnActivateInt[6] := TRUE;
   instKP8Drvs[12].btnActivateInt[7] := TRUE;
   instKP8Drvs[12].btnClrMskOffInt[0] := 16#0000_0000;
   instKP8Drvs[12].btnClrMskOffInt[1] := 16#0002_0000;
   instKP8Drvs[12].btnClrMskOffInt[2] := 16#0004_0000;
   instKP8Drvs[12].btnClrMskOffInt[3] := 16#0008_0000;
   instKP8Drvs[12].btnClrMskOffInt[4] := 16#0000_0000;
   instKP8Drvs[12].btnClrMskOffInt[5] := 16#0020_0000;
   instKP8Drvs[12].btnClrMskOffInt[6] := 16#0040_0000;
   instKP8Drvs[12].btnClrMskOffInt[7] := 16#0080_0000;
   instKP8Drvs[12].btnClrMskOn1Int[0] := 16#0000_0000;
   instKP8Drvs[12].btnClrMskOn1Int[1] := 16#0202_0000;
   instKP8Drvs[12].btnClrMskOn1Int[2] := 16#0404_0000;
   instKP8Drvs[12].btnClrMskOn1Int[3] := 16#0808_0000;
   instKP8Drvs[12].btnClrMskOn1Int[4] := 16#0000_0000;
   instKP8Drvs[12].btnClrMskOn1Int[5] := 16#2020_0000;
   instKP8Drvs[12].btnClrMskOn1Int[6] := 16#4040_0000;
   instKP8Drvs[12].btnClrMskOn1Int[7] := 16#8080_0000;
   instKP8Drvs[12].btnClrMskOn2Int[0] := 16#0000_0000;
   instKP8Drvs[12].btnClrMskOn2Int[1] := 16#0000_0000;
   instKP8Drvs[12].btnClrMskOn2Int[2] := 16#0000_0000;
   instKP8Drvs[12].btnClrMskOn2Int[3] := 16#0000_0000;
   instKP8Drvs[12].btnClrMskOn2Int[4] := 16#0000_0000;
   instKP8Drvs[12].btnClrMskOn2Int[5] := 16#0000_0000;
   instKP8Drvs[12].btnClrMskOn2Int[6] := 16#0000_0000;
   instKP8Drvs[12].btnClrMskOn2Int[7] := 16#0000_0000;
   instKP8Drvs[12].btnClrOffInt[0] := 'off';
   instKP8Drvs[12].btnClrOffInt[1] := 'green';
   instKP8Drvs[12].btnClrOffInt[2] := 'green';
   instKP8Drvs[12].btnClrOffInt[3] := 'green';
   instKP8Drvs[12].btnClrOffInt[4] := 'off';
   instKP8Drvs[12].btnClrOffInt[5] := 'green';
   instKP8Drvs[12].btnClrOffInt[6] := 'green';
   instKP8Drvs[12].btnClrOffInt[7] := 'green';
   instKP8Drvs[12].btnClrOn1Int[0] := 'off';
   instKP8Drvs[12].btnClrOn1Int[1] := 'yellow';
   instKP8Drvs[12].btnClrOn1Int[2] := 'yellow';
   instKP8Drvs[12].btnClrOn1Int[3] := 'yellow';
   instKP8Drvs[12].btnClrOn1Int[4] := 'off';
   instKP8Drvs[12].btnClrOn1Int[5] := 'yellow';
   instKP8Drvs[12].btnClrOn1Int[6] := 'yellow';
   instKP8Drvs[12].btnClrOn1Int[7] := 'yellow';
   instKP8Drvs[12].btnClrOn2Int[0] := 'off';
   instKP8Drvs[12].btnClrOn2Int[4] := 'off';
   instKP8Drvs[12].btnColors := 16#00EE_0000;
   instKP8Drvs[12].btnModeInt[1] := TRUE;
   instKP8Drvs[12].btnModeInt[2] := TRUE;
   instKP8Drvs[12].btnModeInt[3] := TRUE;
   instKP8Drvs[12].btnModeInt[5] := TRUE;
   instKP8Drvs[12].btnModeInt[6] := TRUE;
   instKP8Drvs[12].btnModeInt[7] := TRUE;
   instKP8Drvs[13].btn0ColorOn1 := 'off';
   instKP8Drvs[13].btn0ColorOn2 := 'off';
   instKP8Drvs[13].btn0ColorOff := 'off';
   instKP8Drvs[13].btn1ColorOn1 := 'off';
   instKP8Drvs[13].btn1ColorOn2 := 'off';
   instKP8Drvs[13].btn1ColorOff := 'off';
   instKP8Drvs[13].btn2Activate := TRUE;
   instKP8Drvs[13].btn2Mode := TRUE;
   instKP8Drvs[13].btn2ColorOn1 := 'yellow';
   instKP8Drvs[13].btn2ColorOff := 'green';
   instKP8Drvs[13].btn3Activate := TRUE;
   instKP8Drvs[13].btn3Mode := TRUE;
   instKP8Drvs[13].btn3ColorOn1 := 'yellow';
   instKP8Drvs[13].btn3ColorOff := 'green';
   instKP8Drvs[13].btn4ColorOn1 := 'off';
   instKP8Drvs[13].btn4ColorOn2 := 'off';
   instKP8Drvs[13].btn4ColorOff := 'off';
   instKP8Drvs[13].btn5ColorOn1 := 'off';
   instKP8Drvs[13].btn5ColorOn2 := 'off';
   instKP8Drvs[13].btn5ColorOff := 'off';
   instKP8Drvs[13].btn6Activate := TRUE;
   instKP8Drvs[13].btn6Mode := TRUE;
   instKP8Drvs[13].btn6ColorOn1 := 'yellow';
   instKP8Drvs[13].btn6ColorOff := 'green';
   instKP8Drvs[13].btn7Activate := TRUE;
   instKP8Drvs[13].btn7Mode := TRUE;
   instKP8Drvs[13].btn7ColorOn1 := 'yellow';
   instKP8Drvs[13].btn7ColorOff := 'green';
   instKP8Drvs[13].btnColorsOut := 16#00CC_0000;
   instKP8Drvs[13].i1 := 8;
   instKP8Drvs[13].i2 := 8;
   instKP8Drvs[13].btnActivateInt[2] := TRUE;
   instKP8Drvs[13].btnActivateInt[3] := TRUE;
   instKP8Drvs[13].btnActivateInt[6] := TRUE;
   instKP8Drvs[13].btnActivateInt[7] := TRUE;
   instKP8Drvs[13].btnClrMskOffInt[0] := 16#0000_0000;
   instKP8Drvs[13].btnClrMskOffInt[1] := 16#0000_0000;
   instKP8Drvs[13].btnClrMskOffInt[2] := 16#0004_0000;
   instKP8Drvs[13].btnClrMskOffInt[3] := 16#0008_0000;
   instKP8Drvs[13].btnClrMskOffInt[4] := 16#0000_0000;
   instKP8Drvs[13].btnClrMskOffInt[5] := 16#0000_0000;
   instKP8Drvs[13].btnClrMskOffInt[6] := 16#0040_0000;
   instKP8Drvs[13].btnClrMskOffInt[7] := 16#0080_0000;
   instKP8Drvs[13].btnClrMskOn1Int[0] := 16#0000_0000;
   instKP8Drvs[13].btnClrMskOn1Int[1] := 16#0000_0000;
   instKP8Drvs[13].btnClrMskOn1Int[2] := 16#0404_0000;
   instKP8Drvs[13].btnClrMskOn1Int[3] := 16#0808_0000;
   instKP8Drvs[13].btnClrMskOn1Int[4] := 16#0000_0000;
   instKP8Drvs[13].btnClrMskOn1Int[5] := 16#0000_0000;
   instKP8Drvs[13].btnClrMskOn1Int[6] := 16#4040_0000;
   instKP8Drvs[13].btnClrMskOn1Int[7] := 16#8080_0000;
   instKP8Drvs[13].btnClrMskOn2Int[0] := 16#0000_0000;
   instKP8Drvs[13].btnClrMskOn2Int[1] := 16#0000_0000;
   instKP8Drvs[13].btnClrMskOn2Int[2] := 16#0000_0000;
   instKP8Drvs[13].btnClrMskOn2Int[3] := 16#0000_0000;
   instKP8Drvs[13].btnClrMskOn2Int[4] := 16#0000_0000;
   instKP8Drvs[13].btnClrMskOn2Int[5] := 16#0000_0000;
   instKP8Drvs[13].btnClrMskOn2Int[6] := 16#0000_0000;
   instKP8Drvs[13].btnClrMskOn2Int[7] := 16#0000_0000;
   instKP8Drvs[13].btnClrOffInt[0] := 'off';
   instKP8Drvs[13].btnClrOffInt[1] := 'off';
   instKP8Drvs[13].btnClrOffInt[2] := 'green';
   instKP8Drvs[13].btnClrOffInt[3] := 'green';
   instKP8Drvs[13].btnClrOffInt[4] := 'off';
   instKP8Drvs[13].btnClrOffInt[5] := 'off';
   instKP8Drvs[13].btnClrOffInt[6] := 'green';
   instKP8Drvs[13].btnClrOffInt[7] := 'green';
   instKP8Drvs[13].btnClrOn1Int[0] := 'off';
   instKP8Drvs[13].btnClrOn1Int[1] := 'off';
   instKP8Drvs[13].btnClrOn1Int[2] := 'yellow';
   instKP8Drvs[13].btnClrOn1Int[3] := 'yellow';
   instKP8Drvs[13].btnClrOn1Int[4] := 'off';
   instKP8Drvs[13].btnClrOn1Int[5] := 'off';
   instKP8Drvs[13].btnClrOn1Int[6] := 'yellow';
   instKP8Drvs[13].btnClrOn1Int[7] := 'yellow';
   instKP8Drvs[13].btnClrOn2Int[0] := 'off';
   instKP8Drvs[13].btnClrOn2Int[1] := 'off';
   instKP8Drvs[13].btnClrOn2Int[4] := 'off';
   instKP8Drvs[13].btnClrOn2Int[5] := 'off';
   instKP8Drvs[13].btnColors := 16#00CC_0000;
   instKP8Drvs[13].btnModeInt[2] := TRUE;
   instKP8Drvs[13].btnModeInt[3] := TRUE;
   instKP8Drvs[13].btnModeInt[6] := TRUE;
   instKP8Drvs[13].btnModeInt[7] := TRUE;
   instKP8Drvs[14].btn0ColorOn1 := 'off';
   instKP8Drvs[14].btn0ColorOn2 := 'off';
   instKP8Drvs[14].btn0ColorOff := 'off';
   instKP8Drvs[14].btn1ColorOn1 := 'off';
   instKP8Drvs[14].btn1ColorOn2 := 'off';
   instKP8Drvs[14].btn1ColorOff := 'off';
   instKP8Drvs[14].btn2Activate := TRUE;
   instKP8Drvs[14].btn2Mode := TRUE;
   instKP8Drvs[14].btn2ColorOn1 := 'yellow';
   instKP8Drvs[14].btn2ColorOff := 'green';
   instKP8Drvs[14].btn3Activate := TRUE;
   instKP8Drvs[14].btn3Mode := TRUE;
   instKP8Drvs[14].btn3ColorOn1 := 'yellow';
   instKP8Drvs[14].btn3ColorOff := 'green';
   instKP8Drvs[14].btn4ColorOn1 := 'off';
   instKP8Drvs[14].btn4ColorOn2 := 'off';
   instKP8Drvs[14].btn4ColorOff := 'off';
   instKP8Drvs[14].btn5Activate := TRUE;
   instKP8Drvs[14].btn5Mode := TRUE;
   instKP8Drvs[14].btn5ColorOn1 := 'yellow';
   instKP8Drvs[14].btn5ColorOff := 'green';
   instKP8Drvs[14].btn6Activate := TRUE;
   instKP8Drvs[14].btn6Mode := TRUE;
   instKP8Drvs[14].btn6ColorOn1 := 'yellow';
   instKP8Drvs[14].btn6ColorOff := 'green';
   instKP8Drvs[14].btn7Activate := TRUE;
   instKP8Drvs[14].btn7Mode := TRUE;
   instKP8Drvs[14].btn7ColorOn1 := 'yellow';
   instKP8Drvs[14].btn7ColorOff := 'green';
   instKP8Drvs[14].btnColorsOut := 16#00EC_0000;
   instKP8Drvs[14].i1 := 8;
   instKP8Drvs[14].i2 := 8;
   instKP8Drvs[14].btnActivateInt[2] := TRUE;
   instKP8Drvs[14].btnActivateInt[3] := TRUE;
   instKP8Drvs[14].btnActivateInt[5] := TRUE;
   instKP8Drvs[14].btnActivateInt[6] := TRUE;
   instKP8Drvs[14].btnActivateInt[7] := TRUE;
   instKP8Drvs[14].btnClrMskOffInt[0] := 16#0000_0000;
   instKP8Drvs[14].btnClrMskOffInt[1] := 16#0000_0000;
   instKP8Drvs[14].btnClrMskOffInt[2] := 16#0004_0000;
   instKP8Drvs[14].btnClrMskOffInt[3] := 16#0008_0000;
   instKP8Drvs[14].btnClrMskOffInt[4] := 16#0000_0000;
   instKP8Drvs[14].btnClrMskOffInt[5] := 16#0020_0000;
   instKP8Drvs[14].btnClrMskOffInt[6] := 16#0040_0000;
   instKP8Drvs[14].btnClrMskOffInt[7] := 16#0080_0000;
   instKP8Drvs[14].btnClrMskOn1Int[0] := 16#0000_0000;
   instKP8Drvs[14].btnClrMskOn1Int[1] := 16#0000_0000;
   instKP8Drvs[14].btnClrMskOn1Int[2] := 16#0404_0000;
   instKP8Drvs[14].btnClrMskOn1Int[3] := 16#0808_0000;
   instKP8Drvs[14].btnClrMskOn1Int[4] := 16#0000_0000;
   instKP8Drvs[14].btnClrMskOn1Int[5] := 16#2020_0000;
   instKP8Drvs[14].btnClrMskOn1Int[6] := 16#4040_0000;
   instKP8Drvs[14].btnClrMskOn1Int[7] := 16#8080_0000;
   instKP8Drvs[14].btnClrMskOn2Int[0] := 16#0000_0000;
   instKP8Drvs[14].btnClrMskOn2Int[1] := 16#0000_0000;
   instKP8Drvs[14].btnClrMskOn2Int[2] := 16#0000_0000;
   instKP8Drvs[14].btnClrMskOn2Int[3] := 16#0000_0000;
   instKP8Drvs[14].btnClrMskOn2Int[4] := 16#0000_0000;
   instKP8Drvs[14].btnClrMskOn2Int[5] := 16#0000_0000;
   instKP8Drvs[14].btnClrMskOn2Int[6] := 16#0000_0000;
   instKP8Drvs[14].btnClrMskOn2Int[7] := 16#0000_0000;
   instKP8Drvs[14].btnClrOffInt[0] := 'off';
   instKP8Drvs[14].btnClrOffInt[1] := 'off';
   instKP8Drvs[14].btnClrOffInt[2] := 'green';
   instKP8Drvs[14].btnClrOffInt[3] := 'green';
   instKP8Drvs[14].btnClrOffInt[4] := 'off';
   instKP8Drvs[14].btnClrOffInt[5] := 'green';
   instKP8Drvs[14].btnClrOffInt[6] := 'green';
   instKP8Drvs[14].btnClrOffInt[7] := 'green';
   instKP8Drvs[14].btnClrOn1Int[0] := 'off';
   instKP8Drvs[14].btnClrOn1Int[1] := 'off';
   instKP8Drvs[14].btnClrOn1Int[2] := 'yellow';
   instKP8Drvs[14].btnClrOn1Int[3] := 'yellow';
   instKP8Drvs[14].btnClrOn1Int[4] := 'off';
   instKP8Drvs[14].btnClrOn1Int[5] := 'yellow';
   instKP8Drvs[14].btnClrOn1Int[6] := 'yellow';
   instKP8Drvs[14].btnClrOn1Int[7] := 'yellow';
   instKP8Drvs[14].btnClrOn2Int[0] := 'off';
   instKP8Drvs[14].btnClrOn2Int[1] := 'off';
   instKP8Drvs[14].btnClrOn2Int[4] := 'off';
   instKP8Drvs[14].btnColors := 16#00EC_0000;
   instKP8Drvs[14].btnModeInt[2] := TRUE;
   instKP8Drvs[14].btnModeInt[3] := TRUE;
   instKP8Drvs[14].btnModeInt[5] := TRUE;
   instKP8Drvs[14].btnModeInt[6] := TRUE;
   instKP8Drvs[14].btnModeInt[7] := TRUE;
   instKP8Drvs[15].btn0ColorOn1 := 'off';
   instKP8Drvs[15].btn0ColorOn2 := 'off';
   instKP8Drvs[15].btn0ColorOff := 'off';
   instKP8Drvs[15].btn1Activate := TRUE;
   instKP8Drvs[15].btn1Mode := TRUE;
   instKP8Drvs[15].btn1ColorOn1 := 'yellow';
   instKP8Drvs[15].btn1ColorOff := 'green';
   instKP8Drvs[15].btn2Activate := TRUE;
   instKP8Drvs[15].btn2Mode := TRUE;
   instKP8Drvs[15].btn2ColorOn1 := 'yellow';
   instKP8Drvs[15].btn2ColorOff := 'green';
   instKP8Drvs[15].btn3Activate := TRUE;
   instKP8Drvs[15].btn3Mode := TRUE;
   instKP8Drvs[15].btn3ColorOn1 := 'yellow';
   instKP8Drvs[15].btn3ColorOff := 'green';
   instKP8Drvs[15].btn4ColorOn1 := 'off';
   instKP8Drvs[15].btn4ColorOn2 := 'off';
   instKP8Drvs[15].btn4ColorOff := 'off';
   instKP8Drvs[15].btn5Activate := TRUE;
   instKP8Drvs[15].btn5Mode := TRUE;
   instKP8Drvs[15].btn5ColorOn1 := 'yellow';
   instKP8Drvs[15].btn5ColorOff := 'green';
   instKP8Drvs[15].btn6Activate := TRUE;
   instKP8Drvs[15].btn6Mode := TRUE;
   instKP8Drvs[15].btn6ColorOn1 := 'yellow';
   instKP8Drvs[15].btn6ColorOff := 'green';
   instKP8Drvs[15].btn7Activate := TRUE;
   instKP8Drvs[15].btn7Mode := TRUE;
   instKP8Drvs[15].btn7ColorOn1 := 'yellow';
   instKP8Drvs[15].btn7ColorOff := 'green';
   instKP8Drvs[15].btnColorsOut := 16#00EE_0000;
   instKP8Drvs[15].i1 := 8;
   instKP8Drvs[15].i2 := 8;
   instKP8Drvs[15].btnActivateInt[1] := TRUE;
   instKP8Drvs[15].btnActivateInt[2] := TRUE;
   instKP8Drvs[15].btnActivateInt[3] := TRUE;
   instKP8Drvs[15].btnActivateInt[5] := TRUE;
   instKP8Drvs[15].btnActivateInt[6] := TRUE;
   instKP8Drvs[15].btnActivateInt[7] := TRUE;
   instKP8Drvs[15].btnClrMskOffInt[0] := 16#0000_0000;
   instKP8Drvs[15].btnClrMskOffInt[1] := 16#0002_0000;
   instKP8Drvs[15].btnClrMskOffInt[2] := 16#0004_0000;
   instKP8Drvs[15].btnClrMskOffInt[3] := 16#0008_0000;
   instKP8Drvs[15].btnClrMskOffInt[4] := 16#0000_0000;
   instKP8Drvs[15].btnClrMskOffInt[5] := 16#0020_0000;
   instKP8Drvs[15].btnClrMskOffInt[6] := 16#0040_0000;
   instKP8Drvs[15].btnClrMskOffInt[7] := 16#0080_0000;
   instKP8Drvs[15].btnClrMskOn1Int[0] := 16#0000_0000;
   instKP8Drvs[15].btnClrMskOn1Int[1] := 16#0202_0000;
   instKP8Drvs[15].btnClrMskOn1Int[2] := 16#0404_0000;
   instKP8Drvs[15].btnClrMskOn1Int[3] := 16#0808_0000;
   instKP8Drvs[15].btnClrMskOn1Int[4] := 16#0000_0000;
   instKP8Drvs[15].btnClrMskOn1Int[5] := 16#2020_0000;
   instKP8Drvs[15].btnClrMskOn1Int[6] := 16#4040_0000;
   instKP8Drvs[15].btnClrMskOn1Int[7] := 16#8080_0000;
   instKP8Drvs[15].btnClrMskOn2Int[0] := 16#0000_0000;
   instKP8Drvs[15].btnClrMskOn2Int[1] := 16#0000_0000;
   instKP8Drvs[15].btnClrMskOn2Int[2] := 16#0000_0000;
   instKP8Drvs[15].btnClrMskOn2Int[3] := 16#0000_0000;
   instKP8Drvs[15].btnClrMskOn2Int[4] := 16#0000_0000;
   instKP8Drvs[15].btnClrMskOn2Int[5] := 16#0000_0000;
   instKP8Drvs[15].btnClrMskOn2Int[6] := 16#0000_0000;
   instKP8Drvs[15].btnClrMskOn2Int[7] := 16#0000_0000;
   instKP8Drvs[15].btnClrOffInt[0] := 'off';
   instKP8Drvs[15].btnClrOffInt[1] := 'green';
   instKP8Drvs[15].btnClrOffInt[2] := 'green';
   instKP8Drvs[15].btnClrOffInt[3] := 'green';
   instKP8Drvs[15].btnClrOffInt[4] := 'off';
   instKP8Drvs[15].btnClrOffInt[5] := 'green';
   instKP8Drvs[15].btnClrOffInt[6] := 'green';
   instKP8Drvs[15].btnClrOffInt[7] := 'green';
   instKP8Drvs[15].btnClrOn1Int[0] := 'off';
   instKP8Drvs[15].btnClrOn1Int[1] := 'yellow';
   instKP8Drvs[15].btnClrOn1Int[2] := 'yellow';
   instKP8Drvs[15].btnClrOn1Int[3] := 'yellow';
   instKP8Drvs[15].btnClrOn1Int[4] := 'off';
   instKP8Drvs[15].btnClrOn1Int[5] := 'yellow';
   instKP8Drvs[15].btnClrOn1Int[6] := 'yellow';
   instKP8Drvs[15].btnClrOn1Int[7] := 'yellow';
   instKP8Drvs[15].btnClrOn2Int[0] := 'off';
   instKP8Drvs[15].btnClrOn2Int[4] := 'off';
   instKP8Drvs[15].btnColors := 16#00EE_0000;
   instKP8Drvs[15].btnModeInt[1] := TRUE;
   instKP8Drvs[15].btnModeInt[2] := TRUE;
   instKP8Drvs[15].btnModeInt[3] := TRUE;
   instKP8Drvs[15].btnModeInt[5] := TRUE;
   instKP8Drvs[15].btnModeInt[6] := TRUE;
   instKP8Drvs[15].btnModeInt[7] := TRUE;
   instKP8Drvs[16].btn0ColorOn1 := 'off';
   instKP8Drvs[16].btn0ColorOn2 := 'off';
   instKP8Drvs[16].btn0ColorOff := 'off';
   instKP8Drvs[16].btn1ColorOn1 := 'off';
   instKP8Drvs[16].btn1ColorOn2 := 'off';
   instKP8Drvs[16].btn1ColorOff := 'off';
   instKP8Drvs[16].btn2ColorOn1 := 'off';
   instKP8Drvs[16].btn2ColorOn2 := 'off';
   instKP8Drvs[16].btn2ColorOff := 'off';
   instKP8Drvs[16].btn3Activate := TRUE;
   instKP8Drvs[16].btn3Mode := TRUE;
   instKP8Drvs[16].btn3ColorOn1 := 'yellow';
   instKP8Drvs[16].btn3ColorOff := 'green';
   instKP8Drvs[16].btn4ColorOn1 := 'off';
   instKP8Drvs[16].btn4ColorOn2 := 'off';
   instKP8Drvs[16].btn4ColorOff := 'off';
   instKP8Drvs[16].btn5ColorOn1 := 'off';
   instKP8Drvs[16].btn5ColorOn2 := 'off';
   instKP8Drvs[16].btn5ColorOff := 'off';
   instKP8Drvs[16].btn6ColorOn1 := 'off';
   instKP8Drvs[16].btn6ColorOn2 := 'off';
   instKP8Drvs[16].btn6ColorOff := 'off';
   instKP8Drvs[16].btn7Activate := TRUE;
   instKP8Drvs[16].btn7Mode := TRUE;
   instKP8Drvs[16].btn7ColorOn1 := 'yellow';
   instKP8Drvs[16].btn7ColorOff := 'green';
   instKP8Drvs[16].btnColorsOut := 16#0088_0000;
   instKP8Drvs[16].i1 := 8;
   instKP8Drvs[16].i2 := 8;
   instKP8Drvs[16].btnActivateInt[3] := TRUE;
   instKP8Drvs[16].btnActivateInt[7] := TRUE;
   instKP8Drvs[16].btnClrMskOffInt[0] := 16#0000_0000;
   instKP8Drvs[16].btnClrMskOffInt[1] := 16#0000_0000;
   instKP8Drvs[16].btnClrMskOffInt[2] := 16#0000_0000;
   instKP8Drvs[16].btnClrMskOffInt[3] := 16#0008_0000;
   instKP8Drvs[16].btnClrMskOffInt[4] := 16#0000_0000;
   instKP8Drvs[16].btnClrMskOffInt[5] := 16#0000_0000;
   instKP8Drvs[16].btnClrMskOffInt[6] := 16#0000_0000;
   instKP8Drvs[16].btnClrMskOffInt[7] := 16#0080_0000;
   instKP8Drvs[16].btnClrMskOn1Int[0] := 16#0000_0000;
   instKP8Drvs[16].btnClrMskOn1Int[1] := 16#0000_0000;
   instKP8Drvs[16].btnClrMskOn1Int[2] := 16#0000_0000;
   instKP8Drvs[16].btnClrMskOn1Int[3] := 16#0808_0000;
   instKP8Drvs[16].btnClrMskOn1Int[4] := 16#0000_0000;
   instKP8Drvs[16].btnClrMskOn1Int[5] := 16#0000_0000;
   instKP8Drvs[16].btnClrMskOn1Int[6] := 16#0000_0000;
   instKP8Drvs[16].btnClrMskOn1Int[7] := 16#8080_0000;
   instKP8Drvs[16].btnClrMskOn2Int[0] := 16#0000_0000;
   instKP8Drvs[16].btnClrMskOn2Int[1] := 16#0000_0000;
   instKP8Drvs[16].btnClrMskOn2Int[2] := 16#0000_0000;
   instKP8Drvs[16].btnClrMskOn2Int[3] := 16#0000_0000;
   instKP8Drvs[16].btnClrMskOn2Int[4] := 16#0000_0000;
   instKP8Drvs[16].btnClrMskOn2Int[5] := 16#0000_0000;
   instKP8Drvs[16].btnClrMskOn2Int[6] := 16#0000_0000;
   instKP8Drvs[16].btnClrMskOn2Int[7] := 16#0000_0000;
   instKP8Drvs[16].btnClrOffInt[0] := 'off';
   instKP8Drvs[16].btnClrOffInt[1] := 'off';
   instKP8Drvs[16].btnClrOffInt[2] := 'off';
   instKP8Drvs[16].btnClrOffInt[3] := 'green';
   instKP8Drvs[16].btnClrOffInt[4] := 'off';
   instKP8Drvs[16].btnClrOffInt[5] := 'off';
   instKP8Drvs[16].btnClrOffInt[6] := 'off';
   instKP8Drvs[16].btnClrOffInt[7] := 'green';
   instKP8Drvs[16].btnClrOn1Int[0] := 'off';
   instKP8Drvs[16].btnClrOn1Int[1] := 'off';
   instKP8Drvs[16].btnClrOn1Int[2] := 'off';
   instKP8Drvs[16].btnClrOn1Int[3] := 'yellow';
   instKP8Drvs[16].btnClrOn1Int[4] := 'off';
   instKP8Drvs[16].btnClrOn1Int[5] := 'off';
   instKP8Drvs[16].btnClrOn1Int[6] := 'off';
   instKP8Drvs[16].btnClrOn1Int[7] := 'yellow';
   instKP8Drvs[16].btnClrOn2Int[0] := 'off';
   instKP8Drvs[16].btnClrOn2Int[1] := 'off';
   instKP8Drvs[16].btnClrOn2Int[2] := 'off';
   instKP8Drvs[16].btnClrOn2Int[4] := 'off';
   instKP8Drvs[16].btnClrOn2Int[5] := 'off';
   instKP8Drvs[16].btnClrOn2Int[6] := 'off';
   instKP8Drvs[16].btnColors := 16#0088_0000;
   instKP8Drvs[16].btnModeInt[3] := TRUE;
   instKP8Drvs[16].btnModeInt[7] := TRUE;
   instKP8Drvs[17].btn0ColorOn1 := 'off';
   instKP8Drvs[17].btn0ColorOn2 := 'off';
   instKP8Drvs[17].btn0ColorOff := 'off';
   instKP8Drvs[17].btn1ColorOn1 := 'off';
   instKP8Drvs[17].btn1ColorOn2 := 'off';
   instKP8Drvs[17].btn1ColorOff := 'off';
   instKP8Drvs[17].btn2Activate := TRUE;
   instKP8Drvs[17].btn2Mode := TRUE;
   instKP8Drvs[17].btn2ColorOn1 := 'yellow';
   instKP8Drvs[17].btn2ColorOff := 'green';
   instKP8Drvs[17].btn3Activate := TRUE;
   instKP8Drvs[17].btn3Mode := TRUE;
   instKP8Drvs[17].btn3ColorOn1 := 'yellow';
   instKP8Drvs[17].btn3ColorOff := 'green';
   instKP8Drvs[17].btn4ColorOn1 := 'off';
   instKP8Drvs[17].btn4ColorOn2 := 'off';
   instKP8Drvs[17].btn4ColorOff := 'off';
   instKP8Drvs[17].btn5ColorOn1 := 'off';
   instKP8Drvs[17].btn5ColorOn2 := 'off';
   instKP8Drvs[17].btn5ColorOff := 'off';
   instKP8Drvs[17].btn6Activate := TRUE;
   instKP8Drvs[17].btn6Mode := TRUE;
   instKP8Drvs[17].btn6ColorOn1 := 'yellow';
   instKP8Drvs[17].btn6ColorOff := 'green';
   instKP8Drvs[17].btn7Activate := TRUE;
   instKP8Drvs[17].btn7Mode := TRUE;
   instKP8Drvs[17].btn7ColorOn1 := 'yellow';
   instKP8Drvs[17].btn7ColorOff := 'green';
   instKP8Drvs[17].btnColorsOut := 16#00CC_0000;
   instKP8Drvs[17].i1 := 8;
   instKP8Drvs[17].i2 := 8;
   instKP8Drvs[17].btnActivateInt[2] := TRUE;
   instKP8Drvs[17].btnActivateInt[3] := TRUE;
   instKP8Drvs[17].btnActivateInt[6] := TRUE;
   instKP8Drvs[17].btnActivateInt[7] := TRUE;
   instKP8Drvs[17].btnClrMskOffInt[0] := 16#0000_0000;
   instKP8Drvs[17].btnClrMskOffInt[1] := 16#0000_0000;
   instKP8Drvs[17].btnClrMskOffInt[2] := 16#0004_0000;
   instKP8Drvs[17].btnClrMskOffInt[3] := 16#0008_0000;
   instKP8Drvs[17].btnClrMskOffInt[4] := 16#0000_0000;
   instKP8Drvs[17].btnClrMskOffInt[5] := 16#0000_0000;
   instKP8Drvs[17].btnClrMskOffInt[6] := 16#0040_0000;
   instKP8Drvs[17].btnClrMskOffInt[7] := 16#0080_0000;
   instKP8Drvs[17].btnClrMskOn1Int[0] := 16#0000_0000;
   instKP8Drvs[17].btnClrMskOn1Int[1] := 16#0000_0000;
   instKP8Drvs[17].btnClrMskOn1Int[2] := 16#0404_0000;
   instKP8Drvs[17].btnClrMskOn1Int[3] := 16#0808_0000;
   instKP8Drvs[17].btnClrMskOn1Int[4] := 16#0000_0000;
   instKP8Drvs[17].btnClrMskOn1Int[5] := 16#0000_0000;
   instKP8Drvs[17].btnClrMskOn1Int[6] := 16#4040_0000;
   instKP8Drvs[17].btnClrMskOn1Int[7] := 16#8080_0000;
   instKP8Drvs[17].btnClrMskOn2Int[0] := 16#0000_0000;
   instKP8Drvs[17].btnClrMskOn2Int[1] := 16#0000_0000;
   instKP8Drvs[17].btnClrMskOn2Int[2] := 16#0000_0000;
   instKP8Drvs[17].btnClrMskOn2Int[3] := 16#0000_0000;
   instKP8Drvs[17].btnClrMskOn2Int[4] := 16#0000_0000;
   instKP8Drvs[17].btnClrMskOn2Int[5] := 16#0000_0000;
   instKP8Drvs[17].btnClrMskOn2Int[6] := 16#0000_0000;
   instKP8Drvs[17].btnClrMskOn2Int[7] := 16#0000_0000;
   instKP8Drvs[17].btnClrOffInt[0] := 'off';
   instKP8Drvs[17].btnClrOffInt[1] := 'off';
   instKP8Drvs[17].btnClrOffInt[2] := 'green';
   instKP8Drvs[17].btnClrOffInt[3] := 'green';
   instKP8Drvs[17].btnClrOffInt[4] := 'off';
   instKP8Drvs[17].btnClrOffInt[5] := 'off';
   instKP8Drvs[17].btnClrOffInt[6] := 'green';
   instKP8Drvs[17].btnClrOffInt[7] := 'green';
   instKP8Drvs[17].btnClrOn1Int[0] := 'off';
   instKP8Drvs[17].btnClrOn1Int[1] := 'off';
   instKP8Drvs[17].btnClrOn1Int[2] := 'yellow';
   instKP8Drvs[17].btnClrOn1Int[3] := 'yellow';
   instKP8Drvs[17].btnClrOn1Int[4] := 'off';
   instKP8Drvs[17].btnClrOn1Int[5] := 'off';
   instKP8Drvs[17].btnClrOn1Int[6] := 'yellow';
   instKP8Drvs[17].btnClrOn1Int[7] := 'yellow';
   instKP8Drvs[17].btnClrOn2Int[0] := 'off';
   instKP8Drvs[17].btnClrOn2Int[1] := 'off';
   instKP8Drvs[17].btnClrOn2Int[4] := 'off';
   instKP8Drvs[17].btnClrOn2Int[5] := 'off';
   instKP8Drvs[17].btnColors := 16#00CC_0000;
   instKP8Drvs[17].btnModeInt[2] := TRUE;
   instKP8Drvs[17].btnModeInt[3] := TRUE;
   instKP8Drvs[17].btnModeInt[6] := TRUE;
   instKP8Drvs[17].btnModeInt[7] := TRUE;
   instKP8Drvs[18].btn0ColorOn1 := 'off';
   instKP8Drvs[18].btn0ColorOn2 := 'off';
   instKP8Drvs[18].btn0ColorOff := 'off';
   instKP8Drvs[18].btn1ColorOn1 := 'off';
   instKP8Drvs[18].btn1ColorOn2 := 'off';
   instKP8Drvs[18].btn1ColorOff := 'off';
   instKP8Drvs[18].btn2ColorOn1 := 'off';
   instKP8Drvs[18].btn2ColorOn2 := 'off';
   instKP8Drvs[18].btn2ColorOff := 'off';
   instKP8Drvs[18].btn3Activate := TRUE;
   instKP8Drvs[18].btn3Mode := TRUE;
   instKP8Drvs[18].btn3ColorOn1 := 'yellow';
   instKP8Drvs[18].btn3ColorOff := 'green';
   instKP8Drvs[18].btn4ColorOn1 := 'off';
   instKP8Drvs[18].btn4ColorOn2 := 'off';
   instKP8Drvs[18].btn4ColorOff := 'off';
   instKP8Drvs[18].btn5ColorOn1 := 'off';
   instKP8Drvs[18].btn5ColorOn2 := 'off';
   instKP8Drvs[18].btn5ColorOff := 'off';
   instKP8Drvs[18].btn6Activate := TRUE;
   instKP8Drvs[18].btn6Mode := TRUE;
   instKP8Drvs[18].btn6ColorOn1 := 'yellow';
   instKP8Drvs[18].btn6ColorOff := 'green';
   instKP8Drvs[18].btn7Activate := TRUE;
   instKP8Drvs[18].btn7Mode := TRUE;
   instKP8Drvs[18].btn7ColorOn1 := 'yellow';
   instKP8Drvs[18].btn7ColorOff := 'green';
   instKP8Drvs[18].btnColorsOut := 16#00C8_0000;
   instKP8Drvs[18].i1 := 8;
   instKP8Drvs[18].i2 := 8;
   instKP8Drvs[18].btnActivateInt[3] := TRUE;
   instKP8Drvs[18].btnActivateInt[6] := TRUE;
   instKP8Drvs[18].btnActivateInt[7] := TRUE;
   instKP8Drvs[18].btnClrMskOffInt[0] := 16#0000_0000;
   instKP8Drvs[18].btnClrMskOffInt[1] := 16#0000_0000;
   instKP8Drvs[18].btnClrMskOffInt[2] := 16#0000_0000;
   instKP8Drvs[18].btnClrMskOffInt[3] := 16#0008_0000;
   instKP8Drvs[18].btnClrMskOffInt[4] := 16#0000_0000;
   instKP8Drvs[18].btnClrMskOffInt[5] := 16#0000_0000;
   instKP8Drvs[18].btnClrMskOffInt[6] := 16#0040_0000;
   instKP8Drvs[18].btnClrMskOffInt[7] := 16#0080_0000;
   instKP8Drvs[18].btnClrMskOn1Int[0] := 16#0000_0000;
   instKP8Drvs[18].btnClrMskOn1Int[1] := 16#0000_0000;
   instKP8Drvs[18].btnClrMskOn1Int[2] := 16#0000_0000;
   instKP8Drvs[18].btnClrMskOn1Int[3] := 16#0808_0000;
   instKP8Drvs[18].btnClrMskOn1Int[4] := 16#0000_0000;
   instKP8Drvs[18].btnClrMskOn1Int[5] := 16#0000_0000;
   instKP8Drvs[18].btnClrMskOn1Int[6] := 16#4040_0000;
   instKP8Drvs[18].btnClrMskOn1Int[7] := 16#8080_0000;
   instKP8Drvs[18].btnClrMskOn2Int[0] := 16#0000_0000;
   instKP8Drvs[18].btnClrMskOn2Int[1] := 16#0000_0000;
   instKP8Drvs[18].btnClrMskOn2Int[2] := 16#0000_0000;
   instKP8Drvs[18].btnClrMskOn2Int[3] := 16#0000_0000;
   instKP8Drvs[18].btnClrMskOn2Int[4] := 16#0000_0000;
   instKP8Drvs[18].btnClrMskOn2Int[5] := 16#0000_0000;
   instKP8Drvs[18].btnClrMskOn2Int[6] := 16#0000_0000;
   instKP8Drvs[18].btnClrMskOn2Int[7] := 16#0000_0000;
   instKP8Drvs[18].btnClrOffInt[0] := 'off';
   instKP8Drvs[18].btnClrOffInt[1] := 'off';
   instKP8Drvs[18].btnClrOffInt[2] := 'off';
   instKP8Drvs[18].btnClrOffInt[3] := 'green';
   instKP8Drvs[18].btnClrOffInt[4] := 'off';
   instKP8Drvs[18].btnClrOffInt[5] := 'off';
   instKP8Drvs[18].btnClrOffInt[6] := 'green';
   instKP8Drvs[18].btnClrOffInt[7] := 'green';
   instKP8Drvs[18].btnClrOn1Int[0] := 'off';
   instKP8Drvs[18].btnClrOn1Int[1] := 'off';
   instKP8Drvs[18].btnClrOn1Int[2] := 'off';
   instKP8Drvs[18].btnClrOn1Int[3] := 'yellow';
   instKP8Drvs[18].btnClrOn1Int[4] := 'off';
   instKP8Drvs[18].btnClrOn1Int[5] := 'off';
   instKP8Drvs[18].btnClrOn1Int[6] := 'yellow';
   instKP8Drvs[18].btnClrOn1Int[7] := 'yellow';
   instKP8Drvs[18].btnClrOn2Int[0] := 'off';
   instKP8Drvs[18].btnClrOn2Int[1] := 'off';
   instKP8Drvs[18].btnClrOn2Int[2] := 'off';
   instKP8Drvs[18].btnClrOn2Int[4] := 'off';
   instKP8Drvs[18].btnClrOn2Int[5] := 'off';
   instKP8Drvs[18].btnColors := 16#00C8_0000;
   instKP8Drvs[18].btnModeInt[3] := TRUE;
   instKP8Drvs[18].btnModeInt[6] := TRUE;
   instKP8Drvs[18].btnModeInt[7] := TRUE;
   instKP8Drvs[19].btn0ColorOn1 := 'off';
   instKP8Drvs[19].btn0ColorOn2 := 'off';
   instKP8Drvs[19].btn0ColorOff := 'off';
   instKP8Drvs[19].btn1Activate := TRUE;
   instKP8Drvs[19].btn1Mode := TRUE;
   instKP8Drvs[19].btn1ColorOn1 := 'yellow';
   instKP8Drvs[19].btn1ColorOff := 'green';
   instKP8Drvs[19].btn2Activate := TRUE;
   instKP8Drvs[19].btn2Mode := TRUE;
   instKP8Drvs[19].btn2ColorOn1 := 'yellow';
   instKP8Drvs[19].btn2ColorOff := 'green';
   instKP8Drvs[19].btn3Activate := TRUE;
   instKP8Drvs[19].btn3Mode := TRUE;
   instKP8Drvs[19].btn3ColorOn1 := 'yellow';
   instKP8Drvs[19].btn3ColorOff := 'green';
   instKP8Drvs[19].btn4ColorOn1 := 'off';
   instKP8Drvs[19].btn4ColorOn2 := 'off';
   instKP8Drvs[19].btn4ColorOff := 'off';
   instKP8Drvs[19].btn5Activate := TRUE;
   instKP8Drvs[19].btn5Mode := TRUE;
   instKP8Drvs[19].btn5ColorOn1 := 'yellow';
   instKP8Drvs[19].btn5ColorOff := 'green';
   instKP8Drvs[19].btn6Activate := TRUE;
   instKP8Drvs[19].btn6Mode := TRUE;
   instKP8Drvs[19].btn6ColorOn1 := 'yellow';
   instKP8Drvs[19].btn6ColorOff := 'green';
   instKP8Drvs[19].btn7Activate := TRUE;
   instKP8Drvs[19].btn7Mode := TRUE;
   instKP8Drvs[19].btn7ColorOn1 := 'yellow';
   instKP8Drvs[19].btn7ColorOff := 'green';
   instKP8Drvs[19].btnColorsOut := 16#00EE_0000;
   instKP8Drvs[19].i1 := 8;
   instKP8Drvs[19].i2 := 8;
   instKP8Drvs[19].btnActivateInt[1] := TRUE;
   instKP8Drvs[19].btnActivateInt[2] := TRUE;
   instKP8Drvs[19].btnActivateInt[3] := TRUE;
   instKP8Drvs[19].btnActivateInt[5] := TRUE;
   instKP8Drvs[19].btnActivateInt[6] := TRUE;
   instKP8Drvs[19].btnActivateInt[7] := TRUE;
   instKP8Drvs[19].btnClrMskOffInt[0] := 16#0000_0000;
   instKP8Drvs[19].btnClrMskOffInt[1] := 16#0002_0000;
   instKP8Drvs[19].btnClrMskOffInt[2] := 16#0004_0000;
   instKP8Drvs[19].btnClrMskOffInt[3] := 16#0008_0000;
   instKP8Drvs[19].btnClrMskOffInt[4] := 16#0000_0000;
   instKP8Drvs[19].btnClrMskOffInt[5] := 16#0020_0000;
   instKP8Drvs[19].btnClrMskOffInt[6] := 16#0040_0000;
   instKP8Drvs[19].btnClrMskOffInt[7] := 16#0080_0000;
   instKP8Drvs[19].btnClrMskOn1Int[0] := 16#0000_0000;
   instKP8Drvs[19].btnClrMskOn1Int[1] := 16#0202_0000;
   instKP8Drvs[19].btnClrMskOn1Int[2] := 16#0404_0000;
   instKP8Drvs[19].btnClrMskOn1Int[3] := 16#0808_0000;
   instKP8Drvs[19].btnClrMskOn1Int[4] := 16#0000_0000;
   instKP8Drvs[19].btnClrMskOn1Int[5] := 16#2020_0000;
   instKP8Drvs[19].btnClrMskOn1Int[6] := 16#4040_0000;
   instKP8Drvs[19].btnClrMskOn1Int[7] := 16#8080_0000;
   instKP8Drvs[19].btnClrMskOn2Int[0] := 16#0000_0000;
   instKP8Drvs[19].btnClrMskOn2Int[1] := 16#0000_0000;
   instKP8Drvs[19].btnClrMskOn2Int[2] := 16#0000_0000;
   instKP8Drvs[19].btnClrMskOn2Int[3] := 16#0000_0000;
   instKP8Drvs[19].btnClrMskOn2Int[4] := 16#0000_0000;
   instKP8Drvs[19].btnClrMskOn2Int[5] := 16#0000_0000;
   instKP8Drvs[19].btnClrMskOn2Int[6] := 16#0000_0000;
   instKP8Drvs[19].btnClrMskOn2Int[7] := 16#0000_0000;
   instKP8Drvs[19].btnClrOffInt[0] := 'off';
   instKP8Drvs[19].btnClrOffInt[1] := 'green';
   instKP8Drvs[19].btnClrOffInt[2] := 'green';
   instKP8Drvs[19].btnClrOffInt[3] := 'green';
   instKP8Drvs[19].btnClrOffInt[4] := 'off';
   instKP8Drvs[19].btnClrOffInt[5] := 'green';
   instKP8Drvs[19].btnClrOffInt[6] := 'green';
   instKP8Drvs[19].btnClrOffInt[7] := 'green';
   instKP8Drvs[19].btnClrOn1Int[0] := 'off';
   instKP8Drvs[19].btnClrOn1Int[1] := 'yellow';
   instKP8Drvs[19].btnClrOn1Int[2] := 'yellow';
   instKP8Drvs[19].btnClrOn1Int[3] := 'yellow';
   instKP8Drvs[19].btnClrOn1Int[4] := 'off';
   instKP8Drvs[19].btnClrOn1Int[5] := 'yellow';
   instKP8Drvs[19].btnClrOn1Int[6] := 'yellow';
   instKP8Drvs[19].btnClrOn1Int[7] := 'yellow';
   instKP8Drvs[19].btnClrOn2Int[0] := 'off';
   instKP8Drvs[19].btnClrOn2Int[4] := 'off';
   instKP8Drvs[19].btnColors := 16#00EE_0000;
   instKP8Drvs[19].btnModeInt[1] := TRUE;
   instKP8Drvs[19].btnModeInt[2] := TRUE;
   instKP8Drvs[19].btnModeInt[3] := TRUE;
   instKP8Drvs[19].btnModeInt[5] := TRUE;
   instKP8Drvs[19].btnModeInt[6] := TRUE;
   instKP8Drvs[19].btnModeInt[7] := TRUE;
   instKP8Drvs[20].btn0ColorOn1 := 'off';
   instKP8Drvs[20].btn0ColorOn2 := 'off';
   instKP8Drvs[20].btn0ColorOff := 'off';
   instKP8Drvs[20].btn1ColorOn1 := 'off';
   instKP8Drvs[20].btn1ColorOn2 := 'off';
   instKP8Drvs[20].btn1ColorOff := 'off';
   instKP8Drvs[20].btn2ColorOn1 := 'off';
   instKP8Drvs[20].btn2ColorOn2 := 'off';
   instKP8Drvs[20].btn2ColorOff := 'off';
   instKP8Drvs[20].btn3ColorOn1 := 'off';
   instKP8Drvs[20].btn3ColorOn2 := 'off';
   instKP8Drvs[20].btn3ColorOff := 'off';
   instKP8Drvs[20].btn4ColorOn1 := 'off';
   instKP8Drvs[20].btn4ColorOn2 := 'off';
   instKP8Drvs[20].btn4ColorOff := 'off';
   instKP8Drvs[20].btn5ColorOn1 := 'off';
   instKP8Drvs[20].btn5ColorOn2 := 'off';
   instKP8Drvs[20].btn5ColorOff := 'off';
   instKP8Drvs[20].btn6ColorOn1 := 'off';
   instKP8Drvs[20].btn6ColorOn2 := 'off';
   instKP8Drvs[20].btn6ColorOff := 'off';
   instKP8Drvs[20].btn7ColorOn1 := 'off';
   instKP8Drvs[20].btn7ColorOn2 := 'off';
   instKP8Drvs[20].btn7ColorOff := 'off';
   instKP8Drvs[20].btnColorsOut := 16#0000_0000;
   instKP8Drvs[20].i1 := 8;
   instKP8Drvs[20].btnClrMskOffInt[0] := 16#0000_0000;
   instKP8Drvs[20].btnClrMskOffInt[1] := 16#0000_0000;
   instKP8Drvs[20].btnClrMskOffInt[2] := 16#0000_0000;
   instKP8Drvs[20].btnClrMskOffInt[3] := 16#0000_0000;
   instKP8Drvs[20].btnClrMskOffInt[4] := 16#0000_0000;
   instKP8Drvs[20].btnClrMskOffInt[5] := 16#0000_0000;
   instKP8Drvs[20].btnClrMskOffInt[6] := 16#0000_0000;
   instKP8Drvs[20].btnClrMskOffInt[7] := 16#0000_0000;
   instKP8Drvs[20].btnClrMskOn1Int[0] := 16#0000_0000;
   instKP8Drvs[20].btnClrMskOn1Int[1] := 16#0000_0000;
   instKP8Drvs[20].btnClrMskOn1Int[2] := 16#0000_0000;
   instKP8Drvs[20].btnClrMskOn1Int[3] := 16#0000_0000;
   instKP8Drvs[20].btnClrMskOn1Int[4] := 16#0000_0000;
   instKP8Drvs[20].btnClrMskOn1Int[5] := 16#0000_0000;
   instKP8Drvs[20].btnClrMskOn1Int[6] := 16#0000_0000;
   instKP8Drvs[20].btnClrMskOn1Int[7] := 16#0000_0000;
   instKP8Drvs[20].btnClrMskOn2Int[0] := 16#0000_0000;
   instKP8Drvs[20].btnClrMskOn2Int[1] := 16#0000_0000;
   instKP8Drvs[20].btnClrMskOn2Int[2] := 16#0000_0000;
   instKP8Drvs[20].btnClrMskOn2Int[3] := 16#0000_0000;
   instKP8Drvs[20].btnClrMskOn2Int[4] := 16#0000_0000;
   instKP8Drvs[20].btnClrMskOn2Int[5] := 16#0000_0000;
   instKP8Drvs[20].btnClrMskOn2Int[6] := 16#0000_0000;
   instKP8Drvs[20].btnClrMskOn2Int[7] := 16#0000_0000;
   instKP8Drvs[20].btnClrOffInt[0] := 'off';
   instKP8Drvs[20].btnClrOffInt[1] := 'off';
   instKP8Drvs[20].btnClrOffInt[2] := 'off';
   instKP8Drvs[20].btnClrOffInt[3] := 'off';
   instKP8Drvs[20].btnClrOffInt[4] := 'off';
   instKP8Drvs[20].btnClrOffInt[5] := 'off';
   instKP8Drvs[20].btnClrOffInt[6] := 'off';
   instKP8Drvs[20].btnClrOffInt[7] := 'off';
   instKP8Drvs[20].btnClrOn1Int[0] := 'off';
   instKP8Drvs[20].btnClrOn1Int[1] := 'off';
   instKP8Drvs[20].btnClrOn1Int[2] := 'off';
   instKP8Drvs[20].btnClrOn1Int[3] := 'off';
   instKP8Drvs[20].btnClrOn1Int[4] := 'off';
   instKP8Drvs[20].btnClrOn1Int[5] := 'off';
   instKP8Drvs[20].btnClrOn1Int[6] := 'off';
   instKP8Drvs[20].btnClrOn1Int[7] := 'off';
   instKP8Drvs[20].btnClrOn2Int[0] := 'off';
   instKP8Drvs[20].btnClrOn2Int[1] := 'off';
   instKP8Drvs[20].btnClrOn2Int[2] := 'off';
   instKP8Drvs[20].btnClrOn2Int[3] := 'off';
   instKP8Drvs[20].btnClrOn2Int[4] := 'off';
   instKP8Drvs[20].btnClrOn2Int[5] := 'off';
   instKP8Drvs[20].btnClrOn2Int[6] := 'off';
   instKP8Drvs[20].btnClrOn2Int[7] := 'off';
   instKP8Drvs[20].btnColors := 16#0000_0000;
   instKP8Drvs[21].btn0ColorOn1 := 'off';
   instKP8Drvs[21].btn0ColorOn2 := 'off';
   instKP8Drvs[21].btn0ColorOff := 'off';
   instKP8Drvs[21].btn1ColorOn1 := 'off';
   instKP8Drvs[21].btn1ColorOn2 := 'off';
   instKP8Drvs[21].btn1ColorOff := 'off';
   instKP8Drvs[21].btn2ColorOn1 := 'off';
   instKP8Drvs[21].btn2ColorOn2 := 'off';
   instKP8Drvs[21].btn2ColorOff := 'off';
   instKP8Drvs[21].btn3ColorOn1 := 'off';
   instKP8Drvs[21].btn3ColorOn2 := 'off';
   instKP8Drvs[21].btn3ColorOff := 'off';
   instKP8Drvs[21].btn4ColorOn1 := 'off';
   instKP8Drvs[21].btn4ColorOn2 := 'off';
   instKP8Drvs[21].btn4ColorOff := 'off';
   instKP8Drvs[21].btn5ColorOn1 := 'off';
   instKP8Drvs[21].btn5ColorOn2 := 'off';
   instKP8Drvs[21].btn5ColorOff := 'off';
   instKP8Drvs[21].btn6ColorOn1 := 'off';
   instKP8Drvs[21].btn6ColorOn2 := 'off';
   instKP8Drvs[21].btn6ColorOff := 'off';
   instKP8Drvs[21].btn7Activate := TRUE;
   instKP8Drvs[21].btn7Mode := TRUE;
   instKP8Drvs[21].btn7ColorOn1 := 'yellow';
   instKP8Drvs[21].btn7ColorOff := 'green';
   instKP8Drvs[21].btnColorsOut := 16#0080_0000;
   instKP8Drvs[21].i1 := 8;
   instKP8Drvs[21].i2 := 8;
   instKP8Drvs[21].btnActivateInt[7] := TRUE;
   instKP8Drvs[21].btnClrMskOffInt[0] := 16#0000_0000;
   instKP8Drvs[21].btnClrMskOffInt[1] := 16#0000_0000;
   instKP8Drvs[21].btnClrMskOffInt[2] := 16#0000_0000;
   instKP8Drvs[21].btnClrMskOffInt[3] := 16#0000_0000;
   instKP8Drvs[21].btnClrMskOffInt[4] := 16#0000_0000;
   instKP8Drvs[21].btnClrMskOffInt[5] := 16#0000_0000;
   instKP8Drvs[21].btnClrMskOffInt[6] := 16#0000_0000;
   instKP8Drvs[21].btnClrMskOffInt[7] := 16#0080_0000;
   instKP8Drvs[21].btnClrMskOn1Int[0] := 16#0000_0000;
   instKP8Drvs[21].btnClrMskOn1Int[1] := 16#0000_0000;
   instKP8Drvs[21].btnClrMskOn1Int[2] := 16#0000_0000;
   instKP8Drvs[21].btnClrMskOn1Int[3] := 16#0000_0000;
   instKP8Drvs[21].btnClrMskOn1Int[4] := 16#0000_0000;
   instKP8Drvs[21].btnClrMskOn1Int[5] := 16#0000_0000;
   instKP8Drvs[21].btnClrMskOn1Int[6] := 16#0000_0000;
   instKP8Drvs[21].btnClrMskOn1Int[7] := 16#8080_0000;
   instKP8Drvs[21].btnClrMskOn2Int[0] := 16#0000_0000;
   instKP8Drvs[21].btnClrMskOn2Int[1] := 16#0000_0000;
   instKP8Drvs[21].btnClrMskOn2Int[2] := 16#0000_0000;
   instKP8Drvs[21].btnClrMskOn2Int[3] := 16#0000_0000;
   instKP8Drvs[21].btnClrMskOn2Int[4] := 16#0000_0000;
   instKP8Drvs[21].btnClrMskOn2Int[5] := 16#0000_0000;
   instKP8Drvs[21].btnClrMskOn2Int[6] := 16#0000_0000;
   instKP8Drvs[21].btnClrMskOn2Int[7] := 16#0000_0000;
   instKP8Drvs[21].btnClrOffInt[0] := 'off';
   instKP8Drvs[21].btnClrOffInt[1] := 'off';
   instKP8Drvs[21].btnClrOffInt[2] := 'off';
   instKP8Drvs[21].btnClrOffInt[3] := 'off';
   instKP8Drvs[21].btnClrOffInt[4] := 'off';
   instKP8Drvs[21].btnClrOffInt[5] := 'off';
   instKP8Drvs[21].btnClrOffInt[6] := 'off';
   instKP8Drvs[21].btnClrOffInt[7] := 'green';
   instKP8Drvs[21].btnClrOn1Int[0] := 'off';
   instKP8Drvs[21].btnClrOn1Int[1] := 'off';
   instKP8Drvs[21].btnClrOn1Int[2] := 'off';
   instKP8Drvs[21].btnClrOn1Int[3] := 'off';
   instKP8Drvs[21].btnClrOn1Int[4] := 'off';
   instKP8Drvs[21].btnClrOn1Int[5] := 'off';
   instKP8Drvs[21].btnClrOn1Int[6] := 'off';
   instKP8Drvs[21].btnClrOn1Int[7] := 'yellow';
   instKP8Drvs[21].btnClrOn2Int[0] := 'off';
   instKP8Drvs[21].btnClrOn2Int[1] := 'off';
   instKP8Drvs[21].btnClrOn2Int[2] := 'off';
   instKP8Drvs[21].btnClrOn2Int[3] := 'off';
   instKP8Drvs[21].btnClrOn2Int[4] := 'off';
   instKP8Drvs[21].btnClrOn2Int[5] := 'off';
   instKP8Drvs[21].btnClrOn2Int[6] := 'off';
   instKP8Drvs[21].btnColors := 16#0080_0000;
   instKP8Drvs[21].btnModeInt[7] := TRUE;
   instKP8Drvs[22].btn0ColorOn1 := 'off';
   instKP8Drvs[22].btn0ColorOn2 := 'off';
   instKP8Drvs[22].btn0ColorOff := 'off';
   instKP8Drvs[22].btn1ColorOn1 := 'off';
   instKP8Drvs[22].btn1ColorOn2 := 'off';
   instKP8Drvs[22].btn1ColorOff := 'off';
   instKP8Drvs[22].btn2ColorOn1 := 'off';
   instKP8Drvs[22].btn2ColorOn2 := 'off';
   instKP8Drvs[22].btn2ColorOff := 'off';
   instKP8Drvs[22].btn3Activate := TRUE;
   instKP8Drvs[22].btn3Mode := TRUE;
   instKP8Drvs[22].btn3ColorOn1 := 'yellow';
   instKP8Drvs[22].btn3ColorOff := 'green';
   instKP8Drvs[22].btn4ColorOn1 := 'off';
   instKP8Drvs[22].btn4ColorOn2 := 'off';
